  MoveC 4621 to (-315.82, 6.77, -76.56) mm, rotated rx -179.15 ry 0 rz -30.08 deg; joints [-3.162, -77.655, 137.613, -184.044, 59.828, 242.156] to (-316.49, 5.6, -77.12) mm, rotated rx -179.15 ry 0 rz -30.08 deg; joints [-3.197, -77.547, 137.594, -184.08, 59.918, 242.169]
  MoveL 4622 to (-316.49, 5.6, -77.12) mm, rotated rx -179.15 ry 0 rz -30.08 deg; joints [-3.197, -77.547, 137.594, -184.08, 59.918, 242.169]
  MoveC 4623 to (-316.55, 5.47, -77.12) mm, rotated rx -179.15 ry 0 rz -30.08 deg; joints [-3.2, -77.538, 137.596, -184.083, 59.93, 242.169] to (-316.58, 5.33, -77.12) mm, rotated rx -179.15 ry 0 rz -30.08 deg; joints [-3.201, -77.529, 137.599, -184.084, 59.942, 242.169]
  MoveL 4624 to (-316.58, 5.33, -77.12) mm, rotated rx -179.15 ry 0 rz -30.08 deg; joints [-3.201, -77.529, 137.599, -184.084, 59.942, 242.169]
  MoveC 4625 to (-316.6, 5.18, -77.12) mm, rotated rx -179.15 ry 0 rz -30.08 deg; joints [-3.203, -77.52, 137.602, -184.085, 59.954, 242.169] to (-316.66, 5.05, -77.12) mm, rotated rx -179.15 ry 0 rz -30.08 deg; joints [-3.206, -77.511, 137.604, -184.088, 59.965, 242.17]
  MoveL 4626 to (-316.66, 5.05, -77.12) mm, rotated rx -179.15 ry 0 rz -30.08 deg; joints [-3.206, -77.511, 137.604, -184.088, 59.965, 242.17]
  MoveL 4627 to (-327.16, -13.08, -77.12) mm, rotated rx -179.15 ry 0 rz -30.08 deg; joints [-3.765, -76.293, 137.92, -184.664, 61.515, 242.347]
  MoveC 4628 to (-327.25, -13.19, -77.12) mm, rotated rx -179.15 ry 0 rz -30.08 deg; joints [-3.77, -76.285, 137.921, -184.668, 61.524, 242.349] to (-327.36, -13.29, -77.12) mm, rotated rx -179.15 ry 0 rz -30.08 deg; joints [-3.776, -76.279, 137.923, -184.675, 61.532, 242.351]
  MoveL 4629 to (-327.36, -13.29, -77.12) mm, rotated rx -179.15 ry 0 rz -30.08 deg; joints [-3.776, -76.279, 137.923, -184.675, 61.532, 242.351]
  MoveC 4630 to (-327.47, -13.38, -77.12) mm, rotated rx -179.15 ry 0 rz -30.08 deg; joints [-3.781, -76.272, 137.924, -184.681, 61.54, 242.354] to (-327.55, -13.5, -77.12) mm, rotated rx -179.15 ry 0 rz -30.08 deg; joints [-3.786, -76.264, 137.926, -184.686, 61.55, 242.355]
  MoveL 4631 to (-327.55, -13.5, -77.12) mm, rotated rx -179.15 ry 0 rz -30.08 deg; joints [-3.786, -76.264, 137.926, -184.686, 61.55, 242.355]
  MoveC 4632 to (-328.23, -14.66, -77.67) mm, rotated rx -179.15 ry 0 rz -30.08 deg; joints [-3.82, -76.154, 137.904, -184.721, 61.639, 242.365] to (-328.51, -15.14, -79.02) mm, rotated rx -179.15 ry 0 rz -30.08 deg; joints [-3.83, -76.049, 137.812, -184.732, 61.654, 242.369]
  MoveL 4633 to (-328.51, -15.14, -79.02) mm, rotated rx -179.15 ry 0 rz -30.08 deg; joints [-3.83, -76.049, 137.812, -184.732, 61.654, 242.369]
  MoveL 4634 to (-328.51, -15.14, -81.56) mm, rotated rx -179.15 ry 0 rz -30.08 deg; joints [-3.821, -75.912, 137.626, -184.724, 61.604, 242.369]
  MoveC 4635 to (-328.23, -14.66, -82.91) mm, rotated rx -179.15 ry 0 rz -30.08 deg; joints [-3.802, -75.873, 137.52, -184.705, 61.536, 242.365] to (-327.55, -13.5, -83.46) mm, rotated rx -179.15 ry 0 rz -30.08 deg; joints [-3.764, -75.922, 137.46, -184.667, 61.426, 242.355]
  MoveL 4636 to (-327.55, -13.5, -83.46) mm, rotated rx -179.15 ry 0 rz -30.08 deg; joints [-3.764, -75.922, 137.46, -184.667, 61.426, 242.355]
  MoveC 4637 to (-327.47, -13.38, -83.46) mm, rotated rx -179.15 ry 0 rz -30.08 deg; joints [-3.76, -75.93, 137.458, -184.662, 61.417, 242.353] to (-327.36, -13.29, -83.46) mm, rotated rx -179.15 ry 0 rz -30.08 deg; joints [-3.754, -75.936, 137.457, -184.655, 61.409, 242.351]
  MoveL 4638 to (-327.36, -13.29, -83.46) mm, rotated rx -179.15 ry 0 rz -30.08 deg; joints [-3.754, -75.936, 137.457, -184.655, 61.409, 242.351]
  MoveC 4639 to (-327.25, -13.19, -83.46) mm, rotated rx -179.15 ry 0 rz -30.08 deg; joints [-3.748, -75.943, 137.456, -184.649, 61.401, 242.348] to (-327.16, -13.08, -83.46) mm, rotated rx -179.15 ry 0 rz -30.08 deg; joints [-3.743, -75.951, 137.454, -184.644, 61.391, 242.347]
  MoveL 4640 to (-327.16, -13.08, -83.46) mm, rotated rx -179.15 ry 0 rz -30.08 deg; joints [-3.743, -75.951, 137.454, -184.644, 61.391, 242.347]
  MoveL 4641 to (-316.66, 5.05, -83.46) mm, rotated rx -179.15 ry 0 rz -30.08 deg; joints [-3.187, -77.159, 137.141, -184.072, 59.853, 242.168]
  MoveC 4642 to (-316.6, 5.19, -83.46) mm, rotated rx -179.15 ry 0 rz -30.08 deg; joints [-3.184, -77.167, 137.138, -184.069, 59.842, 242.168] to (-316.58, 5.33, -83.46) mm, rotated rx -179.15 ry 0 rz -30.08 deg; joints [-3.183, -77.177, 137.135, -184.067, 59.83, 242.168]
  MoveL 4643 to (-316.58, 5.33, -83.46) mm, rotated rx -179.15 ry 0 rz -30.08 deg; joints [-3.183, -77.177, 137.135, -184.067, 59.83, 242.168]
  MoveC 4644 to (-316.55, 5.47, -83.46) mm, rotated rx -179.15 ry 0 rz -30.08 deg; joints [-3.181, -77.186, 137.132, -184.066, 59.818, 242.168] to (-316.49, 5.6, -83.46) mm, rotated rx -179.15 ry 0 rz -30.08 deg; joints [-3.178, -77.194, 137.13, -184.063, 59.807, 242.167]
  MoveL 4645 to (-316.49, 5.6, -83.46) mm, rotated rx -179.15 ry 0 rz -30.08 deg; joints [-3.178, -77.194, 137.13, -184.063, 59.807, 242.167]
  MoveC 4646 to (-315.82, 6.77, -84.02) mm, rotated rx -179.15 ry 0 rz -30.08 deg; joints [-3.141, -77.24, 137.068, -184.024, 59.698, 242.154] to (-315.54, 7.25, -85.37) mm, rotated rx -179.15 ry 0 rz -30.08 deg; joints [-3.122, -77.197, 136.96, -184.006, 59.633, 242.149]
  MoveL 4647 to (-315.54, 7.25, -85.37) mm, rotated rx -179.15 ry 0 rz -30.08 deg; joints [-3.122, -77.197, 136.96, -184.006, 59.633, 242.149]
  MoveL 4648 to (-315.54, 7.25, -87.91) mm, rotated rx -179.15 ry 0 rz -30.08 deg; joints [-3.115, -77.056, 136.774, -183.999, 59.588, 242.148]
  MoveC 4649 to (-315.82, 6.77, -89.26) mm, rotated rx -179.15 ry 0 rz -30.08 deg; joints [-3.126, -76.95, 136.685, -184.011, 59.605, 242.153] to (-316.49, 5.6, -89.81) mm, rotated rx -179.15 ry 0 rz -30.08 deg; joints [-3.16, -76.843, 136.665, -184.047, 59.693, 242.166]
  MoveL 4650 to (-316.49, 5.6, -89.81) mm, rotated rx -179.15 ry 0 rz -30.08 deg; joints [-3.16, -76.843, 136.665, -184.047, 59.693, 242.166]
  MoveC 4651 to (-316.55, 5.47, -89.81) mm, rotated rx -179.15 ry 0 rz -30.08 deg; joints [-3.163, -76.835, 136.668, -184.05, 59.704, 242.167] to (-316.58, 5.33, -89.81) mm, rotated rx -179.15 ry 0 rz -30.08 deg; joints [-3.165, -76.826, 136.67, -184.051, 59.716, 242.167]
  MoveL 4652 to (-316.58, 5.33, -89.81) mm, rotated rx -179.15 ry 0 rz -30.08 deg; joints [-3.165, -76.826, 136.67, -184.051, 59.716, 242.167]
  MoveC 4653 to (-316.6, 5.18, -89.81) mm, rotated rx -179.15 ry 0 rz -30.08 deg; joints [-3.166, -76.817, 136.673, -184.052, 59.728, 242.166] to (-316.66, 5.05, -89.81) mm, rotated rx -179.15 ry 0 rz -30.08 deg; joints [-3.169, -76.808, 136.676, -184.055, 59.739, 242.167]
  MoveL 4654 to (-316.66, 5.05, -89.81) mm, rotated rx -179.15 ry 0 rz -30.08 deg; joints [-3.169, -76.808, 136.676, -184.055, 59.739, 242.167]
  MoveL 4655 to (-327.16, -13.08, -89.81) mm, rotated rx -179.15 ry 0 rz -30.08 deg; joints [-3.722, -75.609, 136.987, -184.626, 61.265, 242.347]
  MoveC 4656 to (-327.25, -13.19, -89.81) mm, rotated rx -179.15 ry 0 rz -30.08 deg; joints [-3.727, -75.602, 136.989, -184.63, 61.274, 242.348] to (-327.36, -13.29, -89.81) mm, rotated rx -179.15 ry 0 rz -30.08 deg; joints [-3.732, -75.595, 136.99, -184.637, 61.282, 242.351]
  MoveL 4657 to (-327.36, -13.29, -89.81) mm, rotated rx -179.15 ry 0 rz -30.08 deg; joints [-3.732, -75.595, 136.99, -184.637, 61.282, 242.351]
  MoveC 4658 to (-327.47, -13.38, -89.81) mm, rotated rx -179.15 ry 0 rz -30.08 deg; joints [-3.738, -75.589, 136.991, -184.643, 61.29, 242.353] to (-327.55, -13.5, -89.81) mm, rotated rx -179.15 ry 0 rz -30.08 deg; joints [-3.743, -75.581, 136.993, -184.648, 61.3, 242.355]
  MoveL 4659 to (-327.55, -13.5, -89.81) mm, rotated rx -179.15 ry 0 rz -30.08 deg; joints [-3.743, -75.581, 136.993, -184.648, 61.3, 242.355]
  MoveC 4660 to (-328.23, -14.66, -90.37) mm, rotated rx -179.15 ry 0 rz -30.08 deg; joints [-3.776, -75.473, 136.97, -184.682, 61.387, 242.365] to (-328.51, -15.14, -91.72) mm, rotated rx -179.15 ry 0 rz -30.08 deg; joints [-3.786, -75.368, 136.879, -184.693, 61.4, 242.369]
  MoveL 4661 to (-328.51, -15.14, -91.72) mm, rotated rx -179.15 ry 0 rz -30.08 deg; joints [-3.786, -75.368, 136.879, -184.693, 61.4, 242.369]
  MoveL 4662 to (-328.51, -15.14, -94.26) mm, rotated rx -179.15 ry 0 rz -30.08 deg; joints [-3.778, -75.233, 136.691, -184.686, 61.348, 242.37]
  MoveC 4663 to (-328.23, -14.66, -95.6) mm, rotated rx -179.15 ry 0 rz -30.08 deg; joints [-3.759, -75.193, 136.584, -184.667, 61.28, 242.365] to (-327.55, -13.5, -96.16) mm, rotated rx -179.15 ry 0 rz -30.08 deg; joints [-3.721, -75.241, 136.525, -184.629, 61.171, 242.355]
  MoveL 4664 to (-327.55, -13.5, -96.16) mm, rotated rx -179.15 ry 0 rz -30.08 deg; joints [-3.721, -75.241, 136.525, -184.629, 61.171, 242.355]
  MoveC 4665 to (-327.47, -13.38, -96.16) mm, rotated rx -179.15 ry 0 rz -30.08 deg; joints [-3.717, -75.249, 136.523, -184.624, 61.161, 242.354] to (-327.36, -13.29, -96.16) mm, rotated rx -179.15 ry 0 rz -30.08 deg; joints [-3.711, -75.255, 136.522, -184.618, 61.154, 242.351]
  MoveL 4666 to (-327.36, -13.29, -96.16) mm, rotated rx -179.15 ry 0 rz -30.08 deg; joints [-3.711, -75.255, 136.522, -184.618, 61.154, 242.351]
  MoveC 4667 to (-327.25, -13.19, -96.16) mm, rotated rx -179.15 ry 0 rz -30.08 deg; joints [-3.705, -75.262, 136.52, -184.612, 61.146, 242.349] to (-327.16, -13.08, -96.16) mm, rotated rx -179.15 ry 0 rz -30.08 deg; joints [-3.701, -75.269, 136.519, -184.607, 61.136, 242.347]
  MoveL 4668 to (-327.16, -13.08, -96.16) mm, rotated rx -179.15 ry 0 rz -30.08 deg; joints [-3.701, -75.269, 136.519, -184.607, 61.136, 242.347]
  MoveL 4669 to (-316.66, 5.05, -96.16) mm, rotated rx -179.15 ry 0 rz -30.08 deg; joints [-3.151, -76.459, 136.21, -184.039, 59.622, 242.166]
  MoveC 4670 to (-316.6, 5.19, -96.16) mm, rotated rx -179.15 ry 0 rz -30.08 deg; joints [-3.148, -76.467, 136.207, -184.036, 59.611, 242.166] to (-316.58, 5.33, -96.16) mm, rotated rx -179.15 ry 0 rz -30.08 deg; joints [-3.147, -76.476, 136.204, -184.035, 59.599, 242.166]
  MoveL 4671 to (-316.58, 5.33, -96.16) mm, rotated rx -179.15 ry 0 rz -30.08 deg; joints [-3.147, -76.476, 136.204, -184.035, 59.599, 242.166]
  MoveC 4672 to (-316.55, 5.47, -96.16) mm, rotated rx -179.15 ry 0 rz -30.08 deg; joints [-3.145, -76.485, 136.202, -184.034, 59.587, 242.166] to (-316.49, 5.6, -96.16) mm, rotated rx -179.15 ry 0 rz -30.08 deg; joints [-3.142, -76.494, 136.199, -184.031, 59.576, 242.165]
  MoveL 4673 to (-316.49, 5.6, -96.16) mm, rotated rx -179.15 ry 0 rz -30.08 deg; joints [-3.142, -76.494, 136.199, -184.031, 59.576, 242.165]
  MoveC 4674 to (-315.82, 6.77, -96.72) mm, rotated rx -179.15 ry 0 rz -30.08 deg; joints [-3.105, -76.538, 136.137, -183.993, 59.468, 242.152] to (-315.54, 7.25, -98.07) mm, rotated rx -179.15 ry 0 rz -30.08 deg; joints [-3.087, -76.495, 136.029, -183.974, 59.403, 242.147]
  MoveL 4675 to (-315.54, 7.25, -98.07) mm, rotated rx -179.15 ry 0 rz -30.08 deg; joints [-3.087, -76.495, 136.029, -183.974, 59.403, 242.147]
  MoveL 4676 to (-315.54, 7.25, -100.61) mm, rotated rx -179.15 ry 0 rz -30.08 deg; joints [-3.08, -76.355, 135.842, -183.968, 59.356, 242.146]
  MoveC 4677 to (-315.82, 6.77, -101.95) mm, rotated rx -179.15 ry 0 rz -30.08 deg; joints [-3.091, -76.25, 135.752, -183.98, 59.37, 242.152] to (-316.49, 5.6, -102.51) mm, rotated rx -179.15 ry 0 rz -30.08 deg; joints [-3.125, -76.145, 135.732, -184.015, 59.457, 242.164]
  MoveL 4678 to (-316.49, 5.6, -102.51) mm, rotated rx -179.15 ry 0 rz -30.08 deg; joints [-3.125, -76.145, 135.732, -184.015, 59.457, 242.164]
  MoveC 4679 to (-316.55, 5.47, -102.51) mm, rotated rx -179.15 ry 0 rz -30.08 deg; joints [-3.128, -76.137, 135.734, -184.018, 59.468, 242.165] to (-316.58, 5.33, -102.51) mm, rotated rx -179.15 ry 0 rz -30.08 deg; joints [-3.129, -76.128, 135.737, -184.02, 59.479, 242.165]
  MoveL 4680 to (-316.58, 5.33, -102.51) mm, rotated rx -179.15 ry 0 rz -30.08 deg; joints [-3.129, -76.128, 135.737, -184.02, 59.479, 242.165]
  MoveC 4681 to (-316.6, 5.18, -102.51) mm, rotated rx -179.15 ry 0 rz -30.08 deg; joints [-3.13, -76.119, 135.74, -184.021, 59.491, 242.165] to (-316.66, 5.05, -102.51) mm, rotated rx -179.15 ry 0 rz -30.08 deg; joints [-3.133, -76.11, 135.742, -184.024, 59.502, 242.166]
  MoveL 4682 to (-316.66, 5.05, -102.51) mm, rotated rx -179.15 ry 0 rz -30.08 deg; joints [-3.133, -76.11, 135.742, -184.024, 59.502, 242.166]
  MoveL 4683 to (-327.16, -13.08, -102.51) mm, rotated rx -179.15 ry 0 rz -30.08 deg; joints [-3.68, -74.931, 136.049, -184.589, 61.005, 242.347]
  MoveC 4684 to (-327.25, -13.19, -102.51) mm, rotated rx -179.15 ry 0 rz -30.08 deg; joints [-3.684, -74.923, 136.051, -184.594, 61.015, 242.349] to (-327.36, -13.29, -102.51) mm, rotated rx -179.15 ry 0 rz -30.08 deg; joints [-3.69, -74.917, 136.052, -184.6, 61.023, 242.352]
  MoveL 4685 to (-327.36, -13.29, -102.51) mm, rotated rx -179.15 ry 0 rz -30.08 deg; joints [-3.69, -74.917, 136.052, -184.6, 61.023, 242.352]
  MoveC 4686 to (-327.47, -13.38, -102.51) mm, rotated rx -179.15 ry 0 rz -30.08 deg; joints [-3.696, -74.91, 136.053, -184.606, 61.03, 242.354] to (-327.55, -13.5, -102.51) mm, rotated rx -179.15 ry 0 rz -30.08 deg; joints [-3.7, -74.902, 136.055, -184.611, 61.04, 242.356]
  MoveL 4687 to (-327.55, -13.5, -102.51) mm, rotated rx -179.15 ry 0 rz -30.08 deg; joints [-3.7, -74.902, 136.055, -184.611, 61.04, 242.356]
  MoveC 4688 to (-328.23, -14.66, -103.07) mm, rotated rx -179.15 ry 0 rz -30.08 deg; joints [-3.734, -74.796, 136.032, -184.645, 61.125, 242.366] to (-328.51, -15.14, -104.42) mm, rotated rx -179.15 ry 0 rz -30.08 deg; joints [-3.744, -74.692, 135.94, -184.656, 61.136, 242.371]
  MoveL 4689 to (-328.51, -15.14, -104.42) mm, rotated rx -179.15 ry 0 rz -30.08 deg; joints [-3.744, -74.692, 135.94, -184.656, 61.136, 242.371]
  MoveL 4690 to (-328.51, -15.14, -106.95) mm, rotated rx -179.15 ry 0 rz -30.08 deg; joints [-3.735, -74.558, 135.752, -184.649, 61.082, 242.371]
  MoveC 4691 to (-328.23, -14.66, -108.3) mm, rotated rx -179.15 ry 0 rz -30.08 deg; joints [-3.716, -74.518, 135.644, -184.63, 61.014, 242.367] to (-327.55, -13.5, -108.86) mm, rotated rx -179.15 ry 0 rz -30.08 deg; joints [-3.68, -74.565, 135.585, -184.593, 60.906, 242.356]
  MoveL 4692 to (-327.55, -13.5, -108.86) mm, rotated rx -179.15 ry 0 rz -30.08 deg; joints [-3.68, -74.565, 135.585, -184.593, 60.906, 242.356]
  MoveC 4693 to (-327.47, -13.38, -108.86) mm, rotated rx -179.15 ry 0 rz -30.08 deg; joints [-3.675, -74.572, 135.583, -184.588, 60.897, 242.355] to (-327.36, -13.29, -108.86) mm, rotated rx -179.15 ry 0 rz -30.08 deg; joints [-3.669, -74.579, 135.582, -184.582, 60.889, 242.352]
  MoveL 4694 to (-327.36, -13.29, -108.86) mm, rotated rx -179.15 ry 0 rz -30.08 deg; joints [-3.669, -74.579, 135.582, -184.582, 60.889, 242.352]
  MoveC 4695 to (-327.25, -13.19, -108.86) mm, rotated rx -179.15 ry 0 rz -30.08 deg; joints [-3.664, -74.585, 135.58, -184.576, 60.881, 242.35] to (-327.16, -13.08, -108.86) mm, rotated rx -179.15 ry 0 rz -30.08 deg; joints [-3.659, -74.593, 135.579, -184.571, 60.872, 242.348]
  MoveL 4696 to (-327.16, -13.08, -108.86) mm, rotated rx -179.15 ry 0 rz -30.08 deg; joints [-3.659, -74.593, 135.579, -184.571, 60.872, 242.348]
  MoveL 4697 to (-316.66, 5.05, -108.86) mm, rotated rx -179.15 ry 0 rz -30.08 deg; joints [-3.116, -75.763, 135.273, -184.008, 59.38, 242.165]
  MoveC 4698 to (-316.6, 5.19, -108.86) mm, rotated rx -179.15 ry 0 rz -30.08 deg; joints [-3.113, -75.772, 135.271, -184.005, 59.369, 242.165] to (-316.58, 5.33, -108.86) mm, rotated rx -179.15 ry 0 rz -30.08 deg; joints [-3.112, -75.781, 135.268, -184.004, 59.358, 242.165]
  MoveL 4699 to (-316.58, 5.33, -108.86) mm, rotated rx -179.15 ry 0 rz -30.08 deg; joints [-3.112, -75.781, 135.268, -184.004, 59.358, 242.165]
  MoveC 4700 to (-316.55, 5.47, -108.86) mm, rotated rx -179.15 ry 0 rz -30.08 deg; joints [-3.11, -75.789, 135.266, -184.003, 59.346, 242.165] to (-316.49, 5.6, -108.86) mm, rotated rx -179.15 ry 0 rz -30.08 deg; joints [-3.107, -75.798, 135.263, -184, 59.335, 242.164]
  MoveL 4701 to (-316.49, 5.6, -108.86) mm, rotated rx -179.15 ry 0 rz -30.08 deg; joints [-3.107, -75.798, 135.263, -184, 59.335, 242.164]
  MoveC 4702 to (-315.82, 6.77, -109.42) mm, rotated rx -179.15 ry 0 rz -30.08 deg; joints [-3.071, -75.841, 135.201, -183.962, 59.228, 242.151] to (-315.54, 7.25, -110.76) mm, rotated rx -179.15 ry 0 rz -30.08 deg; joints [-3.053, -75.798, 135.092, -183.944, 59.163, 242.145]
  MoveL 4703 to (-315.54, 7.25, -110.76) mm, rotated rx -179.15 ry 0 rz -30.08 deg; joints [-3.053, -75.798, 135.092, -183.944, 59.163, 242.145]
  MoveL 4704 to (-315.54, 7.25, -113.3) mm, rotated rx -179.15 ry 0 rz -30.08 deg; joints [-3.046, -75.66, 134.905, -183.938, 59.113, 242.145]
  MoveC 4705 to (-315.82, 6.77, -114.65) mm, rotated rx -179.15 ry 0 rz -30.08 deg; joints [-3.057, -75.556, 134.814, -183.95, 59.127, 242.151] to (-316.49, 5.6, -115.21) mm, rotated rx -179.15 ry 0 rz -30.08 deg; joints [-3.09, -75.452, 134.793, -183.985, 59.211, 242.164]
  MoveL 4706 to (-316.49, 5.6, -115.21) mm, rotated rx -179.15 ry 0 rz -30.08 deg; joints [-3.09, -75.452, 134.793, -183.985, 59.211, 242.164]
  MoveC 4707 to (-316.55, 5.47, -115.21) mm, rotated rx -179.15 ry 0 rz -30.08 deg; joints [-3.093, -75.443, 134.796, -183.988, 59.222, 242.165] to (-316.58, 5.33, -115.21) mm, rotated rx -179.15 ry 0 rz -30.08 deg; joints [-3.094, -75.435, 134.798, -183.989, 59.233, 242.164]
  MoveL 4708 to (-316.58, 5.33, -115.21) mm, rotated rx -179.15 ry 0 rz -30.08 deg; joints [-3.094, -75.435, 134.798, -183.989, 59.233, 242.164]
  MoveC 4709 to (-316.6, 5.18, -115.21) mm, rotated rx -179.15 ry 0 rz -30.08 deg; joints [-3.096, -75.426, 134.801, -183.99, 59.245, 242.164] to (-316.66, 5.05, -115.21) mm, rotated rx -179.15 ry 0 rz -30.08 deg; joints [-3.098, -75.418, 134.804, -183.993, 59.256, 242.165]
  MoveL 4710 to (-316.66, 5.05, -115.21) mm, rotated rx -179.15 ry 0 rz -30.08 deg; joints [-3.098, -75.418, 134.804, -183.993, 59.256, 242.165]
  MoveL 4711 to (-327.16, -13.08, -115.21) mm, rotated rx -179.15 ry 0 rz -30.08 deg; joints [-3.639, -74.256, 135.107, -184.554, 60.737, 242.349]
  MoveC 4712 to (-327.25, -13.19, -115.21) mm, rotated rx -179.15 ry 0 rz -30.08 deg; joints [-3.643, -74.248, 135.109, -184.559, 60.746, 242.351] to (-327.36, -13.29, -115.21) mm, rotated rx -179.15 ry 0 rz -30.08 deg; joints [-3.649, -74.242, 135.11, -184.565, 60.754, 242.353]
  MoveL 4713 to (-327.36, -13.29, -115.21) mm, rotated rx -179.15 ry 0 rz -30.08 deg; joints [-3.649, -74.242, 135.11, -184.565, 60.754, 242.353]
  MoveC 4714 to (-327.47, -13.38, -115.21) mm, rotated rx -179.15 ry 0 rz -30.08 deg; joints [-3.655, -74.236, 135.111, -184.571, 60.761, 242.356] to (-327.55, -13.5, -115.21) mm, rotated rx -179.15 ry 0 rz -30.08 deg; joints [-3.659, -74.228, 135.113, -184.576, 60.771, 242.357]
  MoveL 4715 to (-327.55, -13.5, -115.21) mm, rotated rx -179.15 ry 0 rz -30.08 deg; joints [-3.659, -74.228, 135.113, -184.576, 60.771, 242.357]
  MoveC 4716 to (-328.23, -14.66, -115.77) mm, rotated rx -179.15 ry 0 rz -30.08 deg; joints [-3.692, -74.123, 135.089, -184.61, 60.854, 242.368] to (-328.51, -15.14, -117.11) mm, rotated rx -179.15 ry 0 rz -30.08 deg; joints [-3.702, -74.02, 134.996, -184.621, 60.864, 242.373]
  MoveL 4717 to (-328.51, -15.14, -117.11) mm, rotated rx -179.15 ry 0 rz -30.08 deg; joints [-3.702, -74.02, 134.996, -184.621, 60.864, 242.373]
  MoveL 4718 to (-328.51, -15.14, -119.65) mm, rotated rx -179.15 ry 0 rz -30.08 deg; joints [-3.694, -73.887, 134.807, -184.614, 60.808, 242.373]
  MoveC 4719 to (-328.23, -14.66, -121) mm, rotated rx -179.15 ry 0 rz -30.08 deg; joints [-3.675, -73.847, 134.699, -184.595, 60.739, 242.369] to (-327.55, -13.5, -121.56) mm, rotated rx -179.15 ry 0 rz -30.08 deg; joints [-3.639, -73.893, 134.64, -184.558, 60.633, 242.359]
  MoveL 4720 to (-327.55, -13.5, -121.56) mm, rotated rx -179.15 ry 0 rz -30.08 deg; joints [-3.639, -73.893, 134.64, -184.558, 60.633, 242.359]
  MoveC 4721 to (-327.47, -13.38, -121.56) mm, rotated rx -179.15 ry 0 rz -30.08 deg; joints [-3.634, -73.9, 134.638, -184.554, 60.624, 242.357] to (-327.36, -13.29, -121.56) mm, rotated rx -179.15 ry 0 rz -30.08 deg; joints [-3.629, -73.906, 134.637, -184.548, 60.616, 242.354]
  MoveL 4722 to (-327.36, -13.29, -121.56) mm, rotated rx -179.15 ry 0 rz -30.08 deg; joints [-3.629, -73.906, 134.637, -184.548, 60.616, 242.354]
  MoveC 4723 to (-327.25, -13.19, -121.56) mm, rotated rx -179.15 ry 0 rz -30.08 deg; joints [-3.623, -73.913, 134.636, -184.541, 60.608, 242.352] to (-327.16, -13.08, -121.56) mm, rotated rx -179.15 ry 0 rz -30.08 deg; joints [-3.619, -73.92, 134.634, -184.537, 60.599, 242.35]
  MoveL 4724 to (-327.16, -13.08, -121.56) mm, rotated rx -179.15 ry 0 rz -30.08 deg; joints [-3.619, -73.92, 134.634, -184.537, 60.599, 242.35]
  MoveL 4725 to (-316.66, 5.05, -121.56) mm, rotated rx -179.15 ry 0 rz -30.08 deg; joints [-3.081, -75.073, 134.332, -183.979, 59.129, 242.165]
  MoveC 4726 to (-316.6, 5.19, -121.56) mm, rotated rx -179.15 ry 0 rz -30.08 deg; joints [-3.078, -75.081, 134.33, -183.976, 59.118, 242.164] to (-316.58, 5.33, -121.56) mm, rotated rx -179.15 ry 0 rz -30.08 deg; joints [-3.077, -75.09, 134.327, -183.975, 59.107, 242.165]
  MoveL 4727 to (-316.58, 5.33, -121.56) mm, rotated rx -179.15 ry 0 rz -30.08 deg; joints [-3.077, -75.09, 134.327, -183.975, 59.107, 242.165]
  MoveC 4728 to (-316.55, 5.47, -121.56) mm, rotated rx -179.15 ry 0 rz -30.08 deg; joints [-3.076, -75.099, 134.324, -183.973, 59.095, 242.165] to (-316.49, 5.6, -121.56) mm, rotated rx -179.15 ry 0 rz -30.08 deg; joints [-3.073, -75.107, 134.322, -183.971, 59.084, 242.164]
  MoveL 4729 to (-316.49, 5.6, -121.56) mm, rotated rx -179.15 ry 0 rz -30.08 deg; joints [-3.073, -75.107, 134.322, -183.971, 59.084, 242.164]
  MoveC 4730 to (-315.82, 6.77, -122.11) mm, rotated rx -179.15 ry 0 rz -30.08 deg; joints [-3.037, -75.149, 134.26, -183.933, 58.979, 242.151] to (-315.54, 7.25, -123.46) mm, rotated rx -179.15 ry 0 rz -30.08 deg; joints [-3.019, -75.106, 134.151, -183.915, 58.912, 242.145]
  MoveL 4731 to (-315.54, 7.25, -123.46) mm, rotated rx -179.15 ry 0 rz -30.08 deg; joints [-3.019, -75.106, 134.151, -183.915, 58.912, 242.145]
  MoveL 4732 to (-315.54, 7.25, -126) mm, rotated rx -179.15 ry 0 rz -30.08 deg; joints [-3.012, -74.968, 133.962, -183.909, 58.861, 242.145]
  MoveC 4733 to (-315.82, 6.77, -127.35) mm, rotated rx -179.15 ry 0 rz -30.08 deg; joints [-3.023, -74.865, 133.87, -183.921, 58.873, 242.151] to (-316.49, 5.6, -127.91) mm, rotated rx -179.15 ry 0 rz -30.08 deg; joints [-3.056, -74.763, 133.85, -183.956, 58.956, 242.164]
  MoveL 4734 to (-316.49, 5.6, -127.91) mm, rotated rx -179.15 ry 0 rz -30.08 deg; joints [-3.056, -74.763, 133.85, -183.956, 58.956, 242.164]
  MoveC 4735 to (-316.55, 5.47, -127.91) mm, rotated rx -179.15 ry 0 rz -30.08 deg; joints [-3.059, -74.755, 133.852, -183.959, 58.966, 242.165] to (-316.58, 5.33, -127.91) mm, rotated rx -179.15 ry 0 rz -30.08 deg; joints [-3.06, -74.746, 133.855, -183.96, 58.978, 242.165]
  MoveL 4736 to (-316.58, 5.33, -127.91) mm, rotated rx -179.15 ry 0 rz -30.08 deg; joints [-3.06, -74.746, 133.855, -183.96, 58.978, 242.165]
  MoveC 4737 to (-316.6, 5.18, -127.91) mm, rotated rx -179.15 ry 0 rz -30.08 deg; joints [-3.061, -74.737, 133.857, -183.961, 58.989, 242.165] to (-316.66, 5.05, -127.91) mm, rotated rx -179.15 ry 0 rz -30.08 deg; joints [-3.064, -74.729, 133.86, -183.964, 59, 242.166]
  MoveL 4738 to (-316.66, 5.05, -127.91) mm, rotated rx -179.15 ry 0 rz -30.08 deg; joints [-3.064, -74.729, 133.86, -183.964, 59, 242.166]
  MoveL 4739 to (-327.16, -13.08, -127.91) mm, rotated rx -179.15 ry 0 rz -30.08 deg; joints [-3.599, -73.585, 134.159, -184.52, 60.459, 242.352]
  MoveC 4740 to (-327.25, -13.19, -127.91) mm, rotated rx -179.15 ry 0 rz -30.08 deg; joints [-3.603, -73.578, 134.161, -184.525, 60.468, 242.353] to (-327.36, -13.29, -127.91) mm, rotated rx -179.15 ry 0 rz -30.08 deg; joints [-3.609, -73.572, 134.162, -184.531, 60.476, 242.356]
  MoveL 4741 to (-327.36, -13.29, -127.91) mm, rotated rx -179.15 ry 0 rz -30.08 deg; joints [-3.609, -73.572, 134.162, -184.531, 60.476, 242.356]
  MoveC 4742 to (-327.47, -13.38, -127.91) mm, rotated rx -179.15 ry 0 rz -30.08 deg; joints [-3.614, -73.566, 134.164, -184.537, 60.483, 242.358] to (-327.55, -13.5, -127.91) mm, rotated rx -179.15 ry 0 rz -30.08 deg; joints [-3.619, -73.558, 134.165, -184.542, 60.493, 242.36]
  MoveL 4743 to (-327.55, -13.5, -127.91) mm, rotated rx -179.15 ry 0 rz -30.08 deg; joints [-3.619, -73.558, 134.165, -184.542, 60.493, 242.36]
  MoveC 4744 to (-328.23, -14.66, -128.46) mm, rotated rx -179.15 ry 0 rz -30.08 deg; joints [-3.651, -73.454, 134.141, -184.575, 60.574, 242.371] to (-328.51, -15.14, -129.81) mm, rotated rx -179.15 ry 0 rz -30.08 deg; joints [-3.661, -73.352, 134.048, -184.586, 60.582, 242.376]
  MoveL 4745 to (-328.51, -15.14, -129.81) mm, rotated rx -179.15 ry 0 rz -30.08 deg; joints [-3.661, -73.352, 134.048, -184.586, 60.582, 242.376]
  MoveL 4746 to (-328.51, -15.14, -132.35) mm, rotated rx -179.15 ry 0 rz -30.08 deg; joints [-3.653, -73.219, 133.858, -184.58, 60.525, 242.377]
  MoveC 4747 to (-328.23, -14.66, -133.7) mm, rotated rx -179.15 ry 0 rz -30.08 deg; joints [-3.635, -73.18, 133.749, -184.562, 60.456, 242.372] to (-327.55, -13.5, -134.25) mm, rotated rx -179.15 ry 0 rz -30.08 deg; joints [-3.599, -73.224, 133.69, -184.525, 60.351, 242.362]
  MoveL 4748 to (-327.55, -13.5, -134.25) mm, rotated rx -179.15 ry 0 rz -30.08 deg; joints [-3.599, -73.224, 133.69, -184.525, 60.351, 242.362]
  MoveC 4749 to (-327.47, -13.38, -134.25) mm, rotated rx -179.15 ry 0 rz -30.08 deg; joints [-3.594, -73.232, 133.688, -184.52, 60.341, 242.36] to (-327.36, -13.29, -134.25) mm, rotated rx -179.15 ry 0 rz -30.08 deg; joints [-3.589, -73.238, 133.687, -184.514, 60.334, 242.358]
  MoveL 4750 to (-327.36, -13.29, -134.25) mm, rotated rx -179.15 ry 0 rz -30.08 deg; joints [-3.589, -73.238, 133.687, -184.514, 60.334, 242.358]
  MoveC 4751 to (-327.25, -13.19, -134.25) mm, rotated rx -179.15 ry 0 rz -30.08 deg; joints [-3.583, -73.244, 133.686, -184.508, 60.326, 242.355] to (-327.16, -13.08, -134.25) mm, rotated rx -179.15 ry 0 rz -30.08 deg; joints [-3.579, -73.251, 133.684, -184.504, 60.317, 242.353]
  MoveL 4752 to (-327.16, -13.08, -134.25) mm, rotated rx -179.15 ry 0 rz -30.08 deg; joints [-3.579, -73.251, 133.684, -184.504, 60.317, 242.353]
  MoveL 4753 to (-316.66, 5.05, -134.25) mm, rotated rx -179.15 ry 0 rz -30.08 deg; joints [-3.048, -74.387, 133.386, -183.95, 58.868, 242.166]
  MoveC 4754 to (-316.6, 5.19, -134.25) mm, rotated rx -179.15 ry 0 rz -30.08 deg; joints [-3.045, -74.395, 133.384, -183.947, 58.858, 242.165] to (-316.58, 5.33, -134.25) mm, rotated rx -179.15 ry 0 rz -30.08 deg; joints [-3.043, -74.403, 133.381, -183.946, 58.846, 242.165]
  MoveL 4755 to (-316.58, 5.33, -134.25) mm, rotated rx -179.15 ry 0 rz -30.08 deg; joints [-3.043, -74.403, 133.381, -183.946, 58.846, 242.165]
  MoveC 4756 to (-316.55, 5.47, -134.25) mm, rotated rx -179.15 ry 0 rz -30.08 deg; joints [-3.042, -74.412, 133.378, -183.945, 58.835, 242.166] to (-316.49, 5.6, -134.25) mm, rotated rx -179.15 ry 0 rz -30.08 deg; joints [-3.039, -74.42, 133.376, -183.942, 58.824, 242.165]
  MoveL 4757 to (-316.49, 5.6, -134.25) mm, rotated rx -179.15 ry 0 rz -30.08 deg; joints [-3.039, -74.42, 133.376, -183.942, 58.824, 242.165]
  MoveC 4758 to (-315.82, 6.77, -134.81) mm, rotated rx -179.15 ry 0 rz -30.08 deg; joints [-3.004, -74.462, 133.314, -183.905, 58.72, 242.151] to (-315.54, 7.25, -136.16) mm, rotated rx -179.15 ry 0 rz -30.08 deg; joints [-2.986, -74.419, 133.204, -183.887, 58.653, 242.146]
  MoveL 4759 to (-315.54, 7.25, -136.16) mm, rotated rx -179.15 ry 0 rz -30.08 deg; joints [-2.986, -74.419, 133.204, -183.887, 58.653, 242.146]
  MoveL 4760 to (-315.54, 7.25, -138.7) mm, rotated rx -179.15 ry 0 rz -30.08 deg; joints [-2.979, -74.282, 133.014, -183.882, 58.6, 242.146]
  MoveC 4761 to (-315.82, 6.77, -140.05) mm, rotated rx -179.15 ry 0 rz -30.08 deg; joints [-2.99, -74.179, 132.922, -183.894, 58.61, 242.152] to (-316.49, 5.6, -140.6) mm, rotated rx -179.15 ry 0 rz -30.08 deg; joints [-3.023, -74.078, 132.901, -183.928, 58.691, 242.165]
  MoveL 4762 to (-316.49, 5.6, -140.6) mm, rotated rx -179.15 ry 0 rz -30.08 deg; joints [-3.023, -74.078, 132.901, -183.928, 58.691, 242.165]
  MoveC 4763 to (-316.55, 5.47, -140.6) mm, rotated rx -179.15 ry 0 rz -30.08 deg; joints [-3.026, -74.07, 132.903, -183.931, 58.701, 242.166] to (-316.58, 5.33, -140.6) mm, rotated rx -179.15 ry 0 rz -30.08 deg; joints [-3.027, -74.062, 132.906, -183.932, 58.713, 242.166]
  MoveL 4764 to (-316.58, 5.33, -140.6) mm, rotated rx -179.15 ry 0 rz -30.08 deg; joints [-3.027, -74.062, 132.906, -183.932, 58.713, 242.166]
  MoveC 4765 to (-316.6, 5.18, -140.6) mm, rotated rx -179.15 ry 0 rz -30.08 deg; joints [-3.028, -74.053, 132.908, -183.933, 58.724, 242.166] to (-316.66, 5.05, -140.6) mm, rotated rx -179.15 ry 0 rz -30.08 deg; joints [-3.031, -74.045, 132.911, -183.936, 58.734, 242.167]
  MoveL 4766 to (-316.66, 5.05, -140.6) mm, rotated rx -179.15 ry 0 rz -30.08 deg; joints [-3.031, -74.045, 132.911, -183.936, 58.734, 242.167]
  MoveL 4767 to (-327.16, -13.08, -140.6) mm, rotated rx -179.15 ry 0 rz -30.08 deg; joints [-3.559, -72.918, 133.207, -184.488, 60.173, 242.355]
  MoveC 4768 to (-327.25, -13.19, -140.6) mm, rotated rx -179.15 ry 0 rz -30.08 deg; joints [-3.564, -72.911, 133.209, -184.492, 60.182, 242.357] to (-327.36, -13.29, -140.6) mm, rotated rx -179.15 ry 0 rz -30.08 deg; joints [-3.569, -72.905, 133.21, -184.498, 60.19, 242.36]
  MoveL 4769 to (-327.36, -13.29, -140.6) mm, rotated rx -179.15 ry 0 rz -30.08 deg; joints [-3.569, -72.905, 133.21, -184.498, 60.19, 242.36]
  MoveC 4770 to (-327.47, -13.38, -140.6) mm, rotated rx -179.15 ry 0 rz -30.08 deg; joints [-3.575, -72.899, 133.211, -184.504, 60.197, 242.362] to (-327.55, -13.5, -140.6) mm, rotated rx -179.15 ry 0 rz -30.08 deg; joints [-3.579, -72.892, 133.213, -184.509, 60.206, 242.364]
  MoveL 4771 to (-327.55, -13.5, -140.6) mm, rotated rx -179.15 ry 0 rz -30.08 deg; joints [-3.579, -72.892, 133.213, -184.509, 60.206, 242.364]
  MoveC 4772 to (-328.23, -14.66, -141.16) mm, rotated rx -179.15 ry 0 rz -30.08 deg; joints [-3.611, -72.789, 133.188, -184.543, 60.286, 242.375] to (-328.51, -15.14, -142.51) mm, rotated rx -179.15 ry 0 rz -30.08 deg; joints [-3.621, -72.688, 133.094, -184.554, 60.293, 242.38]
  MoveL 4773 to (-328.51, -15.14, -142.51) mm, rotated rx -179.15 ry 0 rz -30.08 deg; joints [-3.621, -72.688, 133.094, -184.554, 60.293, 242.38]
  MoveL 4774 to (-328.51, -15.14, -145.05) mm, rotated rx -179.15 ry 0 rz -30.08 deg; joints [-3.613, -72.556, 132.903, -184.547, 60.234, 242.381]
  MoveC 4775 to (-328.23, -14.66, -146.39) mm, rotated rx -179.15 ry 0 rz -30.08 deg; joints [-3.595, -72.516, 132.794, -184.529, 60.164, 242.377] to (-327.55, -13.5, -146.95) mm, rotated rx -179.15 ry 0 rz -30.08 deg; joints [-3.56, -72.56, 132.735, -184.493, 60.06, 242.366]
  MoveL 4776 to (-327.55, -13.5, -146.95) mm, rotated rx -179.15 ry 0 rz -30.08 deg; joints [-3.56, -72.56, 132.735, -184.493, 60.06, 242.366]
  MoveC 4777 to (-327.47, -13.38, -146.95) mm, rotated rx -179.15 ry 0 rz -30.08 deg; joints [-3.555, -72.567, 132.733, -184.489, 60.051, 242.364] to (-327.36, -13.29, -146.95) mm, rotated rx -179.15 ry 0 rz -30.08 deg; joints [-3.55, -72.573, 132.732, -184.483, 60.043, 242.362]
  MoveL 4778 to (-327.36, -13.29, -146.95) mm, rotated rx -179.15 ry 0 rz -30.08 deg; joints [-3.55, -72.573, 132.732, -184.483, 60.043, 242.362]
  MoveC 4779 to (-327.25, -13.19, -146.95) mm, rotated rx -179.15 ry 0 rz -30.08 deg; joints [-3.544, -72.579, 132.731, -184.477, 60.036, 242.359] to (-327.16, -13.08, -146.95) mm, rotated rx -179.15 ry 0 rz -30.08 deg; joints [-3.54, -72.586, 132.729, -184.472, 60.027, 242.357]
  MoveL 4780 to (-327.16, -13.08, -146.95) mm, rotated rx -179.15 ry 0 rz -30.08 deg; joints [-3.54, -72.586, 132.729, -184.472, 60.027, 242.357]
  MoveL 4781 to (-316.66, 5.05, -146.95) mm, rotated rx -179.15 ry 0 rz -30.08 deg; joints [-3.015, -73.704, 132.434, -183.923, 58.598, 242.168]
  MoveC 4782 to (-316.6, 5.19, -146.95) mm, rotated rx -179.15 ry 0 rz -30.08 deg; joints [-3.012, -73.712, 132.432, -183.92, 58.588, 242.167] to (-316.58, 5.33, -146.95) mm, rotated rx -179.15 ry 0 rz -30.08 deg; joints [-3.011, -73.721, 132.429, -183.919, 58.577, 242.167]
  MoveL 4783 to (-316.58, 5.33, -146.95) mm, rotated rx -179.15 ry 0 rz -30.08 deg; joints [-3.011, -73.721, 132.429, -183.919, 58.577, 242.167]
  MoveC 4784 to (-316.55, 5.47, -146.95) mm, rotated rx -179.15 ry 0 rz -30.08 deg; joints [-3.009, -73.729, 132.427, -183.918, 58.566, 242.167] to (-316.49, 5.6, -146.95) mm, rotated rx -179.15 ry 0 rz -30.08 deg; joints [-3.006, -73.737, 132.424, -183.915, 58.555, 242.166]
  MoveL 4785 to (-316.49, 5.6, -146.95) mm, rotated rx -179.15 ry 0 rz -30.08 deg; joints [-3.006, -73.737, 132.424, -183.915, 58.555, 242.166]
  MoveC 4786 to (-315.82, 6.77, -147.51) mm, rotated rx -179.15 ry 0 rz -30.08 deg; joints [-2.971, -73.778, 132.362, -183.878, 58.451, 242.153] to (-315.54, 7.25, -148.86) mm, rotated rx -179.15 ry 0 rz -30.08 deg; joints [-2.954, -73.735, 132.252, -183.86, 58.384, 242.148]
  MoveL 4787 to (-315.54, 7.25, -148.86) mm, rotated rx -179.15 ry 0 rz -30.08 deg; joints [-2.954, -73.735, 132.252, -183.86, 58.384, 242.148]
  MoveL 4788 to (-315.54, 7.25, -151.4) mm, rotated rx -179.15 ry 0 rz -30.08 deg; joints [-2.947, -73.599, 132.061, -183.855, 58.329, 242.148]
  MoveC 4789 to (-315.82, 6.77, -152.74) mm, rotated rx -179.15 ry 0 rz -30.08 deg; joints [-2.958, -73.497, 131.968, -183.867, 58.338, 242.154] to (-316.49, 5.6, -153.3) mm, rotated rx -179.15 ry 0 rz -30.08 deg; joints [-2.99, -73.397, 131.947, -183.902, 58.417, 242.167]
  MoveL 4790 to (-316.49, 5.6, -153.3) mm, rotated rx -179.15 ry 0 rz -30.08 deg; joints [-2.99, -73.397, 131.947, -183.902, 58.417, 242.167]
  MoveC 4791 to (-316.55, 5.47, -153.3) mm, rotated rx -179.15 ry 0 rz -30.08 deg; joints [-2.993, -73.389, 131.949, -183.905, 58.428, 242.168] to (-316.58, 5.33, -153.3) mm, rotated rx -179.15 ry 0 rz -30.08 deg; joints [-2.994, -73.381, 131.952, -183.906, 58.439, 242.168]
  MoveL 4792 to (-316.58, 5.33, -153.3) mm, rotated rx -179.15 ry 0 rz -30.08 deg; joints [-2.994, -73.381, 131.952, -183.906, 58.439, 242.168]
  MoveC 4793 to (-316.6, 5.18, -153.3) mm, rotated rx -179.15 ry 0 rz -30.08 deg; joints [-2.996, -73.372, 131.954, -183.907, 58.45, 242.168] to (-316.66, 5.05, -153.3) mm, rotated rx -179.15 ry 0 rz -30.08 deg; joints [-2.998, -73.364, 131.957, -183.91, 58.46, 242.169]
  MoveL 4794 to (-316.66, 5.05, -153.3) mm, rotated rx -179.15 ry 0 rz -30.08 deg; joints [-2.998, -73.364, 131.957, -183.91, 58.46, 242.169]
  MoveL 4795 to (-327.16, -13.08, -153.3) mm, rotated rx -179.15 ry 0 rz -30.08 deg; joints [-3.521, -72.255, 132.249, -184.457, 59.878, 242.36]
  MoveC 4796 to (-327.25, -13.19, -153.3) mm, rotated rx -179.15 ry 0 rz -30.08 deg; joints [-3.525, -72.248, 132.251, -184.461, 59.887, 242.361] to (-327.36, -13.29, -153.3) mm, rotated rx -179.15 ry 0 rz -30.08 deg; joints [-3.531, -72.242, 132.252, -184.467, 59.895, 242.364]
  MoveL 4797 to (-327.36, -13.29, -153.3) mm, rotated rx -179.15 ry 0 rz -30.08 deg; joints [-3.531, -72.242, 132.252, -184.467, 59.895, 242.364]
  MoveC 4798 to (-327.47, -13.38, -153.3) mm, rotated rx -179.15 ry 0 rz -30.08 deg; joints [-3.536, -72.236, 132.253, -184.473, 59.902, 242.367] to (-327.55, -13.5, -153.3) mm, rotated rx -179.15 ry 0 rz -30.08 deg; joints [-3.54, -72.228, 132.255, -184.478, 59.911, 242.368]
  MoveL 4799 to (-327.55, -13.5, -153.3) mm, rotated rx -179.15 ry 0 rz -30.08 deg; joints [-3.54, -72.228, 132.255, -184.478, 59.911, 242.368]
  MoveC 4800 to (-328.23, -14.66, -153.86) mm, rotated rx -179.15 ry 0 rz -30.08 deg; joints [-3.572, -72.127, 132.23, -184.511, 59.989, 242.38] to (-328.51, -15.14, -155.21) mm, rotated rx -179.15 ry 0 rz -30.08 deg; joints [-3.582, -72.027, 132.135, -184.522, 59.994, 242.385]
  MoveL 4801 to (-328.51, -15.14, -155.21) mm, rotated rx -179.15 ry 0 rz -30.08 deg; joints [-3.582, -72.027, 132.135, -184.522, 59.994, 242.385]
  MoveL 4802 to (-328.51, -15.14, -157.74) mm, rotated rx -179.15 ry 0 rz -30.08 deg; joints [-3.574, -71.895, 131.943, -184.516, 59.934, 242.386]
  MoveC 4803 to (-328.23, -14.66, -159.09) mm, rotated rx -179.15 ry 0 rz -30.08 deg; joints [-3.557, -71.855, 131.834, -184.498, 59.864, 242.382] to (-327.55, -13.5, -159.65) mm, rotated rx -179.15 ry 0 rz -30.08 deg; joints [-3.521, -71.898, 131.774, -184.463, 59.76, 242.371]
  MoveL 4804 to (-327.55, -13.5, -159.65) mm, rotated rx -179.15 ry 0 rz -30.08 deg; joints [-3.521, -71.898, 131.774, -184.463, 59.76, 242.371]
  MoveC 4805 to (-327.47, -13.38, -159.65) mm, rotated rx -179.15 ry 0 rz -30.08 deg; joints [-3.517, -71.905, 131.773, -184.458, 59.752, 242.369] to (-327.36, -13.29, -159.65) mm, rotated rx -179.15 ry 0 rz -30.08 deg; joints [-3.512, -71.911, 131.771, -184.452, 59.744, 242.367]
  MoveL 4806 to (-327.36, -13.29, -159.65) mm, rotated rx -179.15 ry 0 rz -30.08 deg; joints [-3.512, -71.911, 131.771, -184.452, 59.744, 242.367]
  MoveC 4807 to (-327.25, -13.19, -159.65) mm, rotated rx -179.15 ry 0 rz -30.08 deg; joints [-3.506, -71.917, 131.77, -184.446, 59.737, 242.364] to (-327.16, -13.08, -159.65) mm, rotated rx -179.15 ry 0 rz -30.08 deg; joints [-3.502, -71.924, 131.769, -184.441, 59.728, 242.362]
  MoveL 4808 to (-327.16, -13.08, -159.65) mm, rotated rx -179.15 ry 0 rz -30.08 deg; joints [-3.502, -71.924, 131.769, -184.441, 59.728, 242.362]
  MoveL 4809 to (-316.66, 5.05, -159.65) mm, rotated rx -179.15 ry 0 rz -30.08 deg; joints [-2.982, -73.025, 131.477, -183.897, 58.32, 242.171]
  MoveC 4810 to (-316.6, 5.19, -159.65) mm, rotated rx -179.15 ry 0 rz -30.08 deg; joints [-2.98, -73.033, 131.475, -183.894, 58.309, 242.17] to (-316.58, 5.33, -159.65) mm, rotated rx -179.15 ry 0 rz -30.08 deg; joints [-2.978, -73.042, 131.472, -183.893, 58.298, 242.17]
  MoveL 4811 to (-316.58, 5.33, -159.65) mm, rotated rx -179.15 ry 0 rz -30.08 deg; joints [-2.978, -73.042, 131.472, -183.893, 58.298, 242.17]
  MoveC 4812 to (-316.55, 5.47, -159.65) mm, rotated rx -179.15 ry 0 rz -30.08 deg; joints [-2.977, -73.05, 131.47, -183.892, 58.287, 242.17] to (-316.49, 5.6, -159.65) mm, rotated rx -179.15 ry 0 rz -30.08 deg; joints [-2.974, -73.058, 131.467, -183.889, 58.277, 242.169]
  MoveL 4813 to (-316.49, 5.6, -159.65) mm, rotated rx -179.15 ry 0 rz -30.08 deg; joints [-2.974, -73.058, 131.467, -183.889, 58.277, 242.169]
  MoveC 4814 to (-315.82, 6.77, -160.21) mm, rotated rx -179.15 ry 0 rz -30.08 deg; joints [-2.939, -73.098, 131.405, -183.852, 58.174, 242.156] to (-315.54, 7.25, -161.55) mm, rotated rx -179.15 ry 0 rz -30.08 deg; joints [-2.922, -73.055, 131.295, -183.835, 58.107, 242.15]
  MoveL 4815 to (-315.54, 7.25, -161.55) mm, rotated rx -179.15 ry 0 rz -30.08 deg; joints [-2.922, -73.055, 131.295, -183.835, 58.107, 242.15]
  MoveL 4816 to (-315.54, 7.25, -164.09) mm, rotated rx -179.15 ry 0 rz -30.08 deg; joints [-2.916, -72.919, 131.103, -183.83, 58.05, 242.151]
  MoveC 4817 to (-315.82, 6.77, -165.44) mm, rotated rx -179.15 ry 0 rz -30.08 deg; joints [-2.927, -72.818, 131.009, -183.842, 58.057, 242.157] to (-316.49, 5.6, -166) mm, rotated rx -179.15 ry 0 rz -30.08 deg; joints [-2.958, -72.72, 130.987, -183.876, 58.135, 242.17]
  MoveL 4818 to (-316.49, 5.6, -166) mm, rotated rx -179.15 ry 0 rz -30.08 deg; joints [-2.958, -72.72, 130.987, -183.876, 58.135, 242.17]
  MoveC 4819 to (-316.55, 5.47, -166) mm, rotated rx -179.15 ry 0 rz -30.08 deg; joints [-2.961, -72.712, 130.989, -183.879, 58.145, 242.171] to (-316.58, 5.33, -166) mm, rotated rx -179.15 ry 0 rz -30.08 deg; joints [-2.963, -72.703, 130.992, -183.88, 58.156, 242.171]
  MoveL 4820 to (-316.58, 5.33, -166) mm, rotated rx -179.15 ry 0 rz -30.08 deg; joints [-2.963, -72.703, 130.992, -183.88, 58.156, 242.171]
  MoveC 4821 to (-316.6, 5.18, -166) mm, rotated rx -179.15 ry 0 rz -30.08 deg; joints [-2.964, -72.695, 130.995, -183.881, 58.167, 242.171] to (-316.66, 5.05, -166) mm, rotated rx -179.15 ry 0 rz -30.08 deg; joints [-2.967, -72.687, 130.997, -183.884, 58.177, 242.172]
  MoveL 4822 to (-316.66, 5.05, -166) mm, rotated rx -179.15 ry 0 rz -30.08 deg; joints [-2.967, -72.687, 130.997, -183.884, 58.177, 242.172]
  MoveL 4823 to (-327.16, -13.08, -166) mm, rotated rx -179.15 ry 0 rz -30.08 deg; joints [-3.483, -71.594, 131.286, -184.427, 59.576, 242.365]
  MoveC 4824 to (-327.25, -13.19, -166) mm, rotated rx -179.15 ry 0 rz -30.08 deg; joints [-3.488, -71.587, 131.288, -184.431, 59.584, 242.367] to (-327.36, -13.29, -166) mm, rotated rx -179.15 ry 0 rz -30.08 deg; joints [-3.493, -71.581, 131.289, -184.437, 59.592, 242.369]
  MoveL 4825 to (-327.36, -13.29, -166) mm, rotated rx -179.15 ry 0 rz -30.08 deg; joints [-3.493, -71.581, 131.289, -184.437, 59.592, 242.369]
  MoveC 4826 to (-327.47, -13.38, -166) mm, rotated rx -179.15 ry 0 rz -30.08 deg; joints [-3.498, -71.575, 131.29, -184.443, 59.599, 242.372] to (-327.55, -13.5, -166) mm, rotated rx -179.15 ry 0 rz -30.08 deg; joints [-3.503, -71.568, 131.292, -184.448, 59.608, 242.374]
  MoveL 4827 to (-327.55, -13.5, -166) mm, rotated rx -179.15 ry 0 rz -30.08 deg; joints [-3.503, -71.568, 131.292, -184.448, 59.608, 242.374]
  MoveC 4828 to (-328.23, -14.66, -166.56) mm, rotated rx -179.15 ry 0 rz -30.08 deg; joints [-3.534, -71.468, 131.267, -184.481, 59.684, 242.385] to (-328.51, -15.14, -167.9) mm, rotated rx -179.15 ry 0 rz -30.08 deg; joints [-3.544, -71.368, 131.171, -184.492, 59.688, 242.39]
  MoveL 4829 to (-328.51, -15.14, -167.9) mm, rotated rx -179.15 ry 0 rz -30.08 deg; joints [-3.544, -71.368, 131.171, -184.492, 59.688, 242.39]
  MoveL 4830 to (-328.51, -15.14, -170.44) mm, rotated rx -179.15 ry 0 rz -30.08 deg; joints [-3.536, -71.237, 130.978, -184.486, 59.626, 242.392]
  MoveC 4831 to (-328.23, -14.66, -171.79) mm, rotated rx -179.15 ry 0 rz -30.08 deg; joints [-3.519, -71.197, 130.868, -184.469, 59.556, 242.388] to (-327.55, -13.5, -172.35) mm, rotated rx -179.15 ry 0 rz -30.08 deg; joints [-3.484, -71.239, 130.809, -184.433, 59.453, 242.377]
  MoveL 4832 to (-327.55, -13.5, -172.35) mm, rotated rx -179.15 ry 0 rz -30.08 deg; joints [-3.484, -71.239, 130.809, -184.433, 59.453, 242.377]
  MoveC 4833 to (-327.47, -13.38, -172.35) mm, rotated rx -179.15 ry 0 rz -30.08 deg; joints [-3.48, -71.246, 130.807, -184.429, 59.444, 242.375] to (-327.36, -13.29, -172.35) mm, rotated rx -179.15 ry 0 rz -30.08 deg; joints [-3.474, -71.252, 130.806, -184.423, 59.437, 242.372]
  MoveL 4834 to (-327.36, -13.29, -172.35) mm, rotated rx -179.15 ry 0 rz -30.08 deg; joints [-3.474, -71.252, 130.806, -184.423, 59.437, 242.372]
  MoveC 4835 to (-327.25, -13.19, -172.35) mm, rotated rx -179.15 ry 0 rz -30.08 deg; joints [-3.469, -71.258, 130.805, -184.417, 59.43, 242.37] to (-327.16, -13.08, -172.35) mm, rotated rx -179.15 ry 0 rz -30.08 deg; joints [-3.465, -71.265, 130.803, -184.412, 59.421, 242.368]
  MoveL 4836 to (-327.16, -13.08, -172.35) mm, rotated rx -179.15 ry 0 rz -30.08 deg; joints [-3.465, -71.265, 130.803, -184.412, 59.421, 242.368]
  MoveL 4837 to (-316.66, 5.05, -172.35) mm, rotated rx -179.15 ry 0 rz -30.08 deg; joints [-2.951, -72.35, 130.515, -183.872, 58.032, 242.174]
  MoveC 4838 to (-316.6, 5.19, -172.35) mm, rotated rx -179.15 ry 0 rz -30.08 deg; joints [-2.948, -72.358, 130.513, -183.869, 58.022, 242.173] to (-316.58, 5.33, -172.35) mm, rotated rx -179.15 ry 0 rz -30.08 deg; joints [-2.947, -72.366, 130.51, -183.868, 58.011, 242.173]
  MoveL 4839 to (-316.58, 5.33, -172.35) mm, rotated rx -179.15 ry 0 rz -30.08 deg; joints [-2.947, -72.366, 130.51, -183.868, 58.011, 242.173]
  MoveC 4840 to (-316.55, 5.47, -172.35) mm, rotated rx -179.15 ry 0 rz -30.08 deg; joints [-2.946, -72.374, 130.507, -183.867, 58, 242.173] to (-316.49, 5.6, -172.35) mm, rotated rx -179.15 ry 0 rz -30.08 deg; joints [-2.943, -72.382, 130.505, -183.864, 57.99, 242.172]
  MoveL 4841 to (-316.49, 5.6, -172.35) mm, rotated rx -179.15 ry 0 rz -30.08 deg; joints [-2.943, -72.382, 130.505, -183.864, 57.99, 242.172]
  MoveC 4842 to (-315.82, 6.77, -172.9) mm, rotated rx -179.15 ry 0 rz -30.08 deg; joints [-2.908, -72.421, 130.443, -183.828, 57.888, 242.159] to (-315.54, 7.25, -174.25) mm, rotated rx -179.15 ry 0 rz -30.08 deg; joints [-2.891, -72.378, 130.332, -183.81, 57.82, 242.154]
  MoveL 4843 to (-315.54, 7.25, -174.25) mm, rotated rx -179.15 ry 0 rz -30.08 deg; joints [-2.891, -72.378, 130.332, -183.81, 57.82, 242.154]
  MoveL 4844 to (-315.54, 7.25, -176.79) mm, rotated rx -179.15 ry 0 rz -30.08 deg; joints [-2.885, -72.243, 130.139, -183.806, 57.762, 242.154]
  MoveC 4845 to (-315.82, 6.77, -178.14) mm, rotated rx -179.15 ry 0 rz -30.08 deg; joints [-2.896, -72.143, 130.045, -183.818, 57.768, 242.16] to (-316.49, 5.6, -178.7) mm, rotated rx -179.15 ry 0 rz -30.08 deg; joints [-2.927, -72.045, 130.022, -183.852, 57.844, 242.174]
  MoveL 4846 to (-316.49, 5.6, -178.7) mm, rotated rx -179.15 ry 0 rz -30.08 deg; joints [-2.927, -72.045, 130.022, -183.852, 57.844, 242.174]
  MoveC 4847 to (-316.55, 5.47, -178.7) mm, rotated rx -179.15 ry 0 rz -30.08 deg; joints [-2.93, -72.037, 130.024, -183.855, 57.854, 242.175] to (-316.58, 5.33, -178.7) mm, rotated rx -179.15 ry 0 rz -30.08 deg; joints [-2.931, -72.029, 130.027, -183.856, 57.864, 242.175]
  MoveL 4848 to (-316.58, 5.33, -178.7) mm, rotated rx -179.15 ry 0 rz -30.08 deg; joints [-2.931, -72.029, 130.027, -183.856, 57.864, 242.175]
  MoveC 4849 to (-316.6, 5.18, -178.7) mm, rotated rx -179.15 ry 0 rz -30.08 deg; joints [-2.933, -72.021, 130.029, -183.857, 57.875, 242.175] to (-316.66, 5.05, -178.7) mm, rotated rx -179.15 ry 0 rz -30.08 deg; joints [-2.935, -72.013, 130.032, -183.86, 57.885, 242.176]
  MoveL 4850 to (-316.66, 5.05, -178.7) mm, rotated rx -179.15 ry 0 rz -30.08 deg; joints [-2.935, -72.013, 130.032, -183.86, 57.885, 242.176]
  MoveL 4851 to (-327.16, -13.08, -178.7) mm, rotated rx -179.15 ry 0 rz -30.08 deg; joints [-3.447, -70.936, 130.318, -184.398, 59.265, 242.371]
  MoveC 4852 to (-327.25, -13.19, -178.7) mm, rotated rx -179.15 ry 0 rz -30.08 deg; joints [-3.451, -70.929, 130.32, -184.403, 59.273, 242.373] to (-327.36, -13.29, -178.7) mm, rotated rx -179.15 ry 0 rz -30.08 deg; joints [-3.456, -70.923, 130.321, -184.409, 59.281, 242.376]
  MoveL 4853 to (-327.36, -13.29, -178.7) mm, rotated rx -179.15 ry 0 rz -30.08 deg; joints [-3.456, -70.923, 130.321, -184.409, 59.281, 242.376]
  MoveC 4854 to (-327.47, -13.38, -178.7) mm, rotated rx -179.15 ry 0 rz -30.08 deg; joints [-3.461, -70.917, 130.322, -184.414, 59.288, 242.378] to (-327.55, -13.5, -178.7) mm, rotated rx -179.15 ry 0 rz -30.08 deg; joints [-3.466, -70.91, 130.324, -184.419, 59.297, 242.38]
  MoveL 4855 to (-327.55, -13.5, -178.7) mm, rotated rx -179.15 ry 0 rz -30.08 deg; joints [-3.466, -70.91, 130.324, -184.419, 59.297, 242.38]
  MoveC 4856 to (-328.23, -14.66, -179.25) mm, rotated rx -179.15 ry 0 rz -30.08 deg; joints [-3.497, -70.811, 130.298, -184.452, 59.371, 242.392] to (-328.51, -15.14, -180.6) mm, rotated rx -179.15 ry 0 rz -30.08 deg; joints [-3.507, -70.713, 130.202, -184.463, 59.374, 242.397]
  MoveL 4857 to (-328.51, -15.14, -180.6) mm, rotated rx -179.15 ry 0 rz -30.08 deg; joints [-3.507, -70.713, 130.202, -184.463, 59.374, 242.397]
  MoveL 4858 to (-328.51, -15.14, -183.14) mm, rotated rx -179.15 ry 0 rz -30.08 deg; joints [-3.499, -70.582, 130.008, -184.457, 59.31, 242.398]
  MoveC 4859 to (-328.23, -14.66, -184.49) mm, rotated rx -179.15 ry 0 rz -30.08 deg; joints [-3.482, -70.542, 129.897, -184.44, 59.24, 242.394] to (-327.55, -13.5, -185.04) mm, rotated rx -179.15 ry 0 rz -30.08 deg; joints [-3.447, -70.583, 129.837, -184.405, 59.138, 242.383]
  MoveL 4860 to (-327.55, -13.5, -185.04) mm, rotated rx -179.15 ry 0 rz -30.08 deg; joints [-3.447, -70.583, 129.837, -184.405, 59.138, 242.383]
  MoveC 4861 to (-327.47, -13.38, -185.04) mm, rotated rx -179.15 ry 0 rz -30.08 deg; joints [-3.443, -70.59, 129.836, -184.401, 59.129, 242.381] to (-327.36, -13.29, -185.04) mm, rotated rx -179.15 ry 0 rz -30.08 deg; joints [-3.438, -70.595, 129.835, -184.395, 59.122, 242.379]
  MoveL 4862 to (-327.36, -13.29, -185.04) mm, rotated rx -179.15 ry 0 rz -30.08 deg; joints [-3.438, -70.595, 129.835, -184.395, 59.122, 242.379]
  MoveC 4863 to (-327.25, -13.19, -185.04) mm, rotated rx -179.15 ry 0 rz -30.08 deg; joints [-3.433, -70.601, 129.834, -184.389, 59.115, 242.376] to (-327.16, -13.08, -185.04) mm, rotated rx -179.15 ry 0 rz -30.08 deg; joints [-3.428, -70.608, 129.832, -184.384, 59.106, 242.375]
  MoveL 4864 to (-327.16, -13.08, -185.04) mm, rotated rx -179.15 ry 0 rz -30.08 deg; joints [-3.428, -70.608, 129.832, -184.384, 59.106, 242.375]
  MoveL 4865 to (-316.66, 5.05, -185.04) mm, rotated rx -179.15 ry 0 rz -30.08 deg; joints [-2.92, -71.678, 129.547, -183.848, 57.736, 242.178]
  MoveC 4866 to (-316.6, 5.19, -185.04) mm, rotated rx -179.15 ry 0 rz -30.08 deg; joints [-2.917, -71.685, 129.545, -183.845, 57.726, 242.177] to (-316.58, 5.33, -185.04) mm, rotated rx -179.15 ry 0 rz -30.08 deg; joints [-2.916, -71.693, 129.542, -183.844, 57.716, 242.177]
  MoveL 4867 to (-316.58, 5.33, -185.04) mm, rotated rx -179.15 ry 0 rz -30.08 deg; joints [-2.916, -71.693, 129.542, -183.844, 57.716, 242.177]
  MoveC 4868 to (-316.55, 5.47, -185.04) mm, rotated rx -179.15 ry 0 rz -30.08 deg; joints [-2.915, -71.701, 129.539, -183.843, 57.705, 242.177] to (-316.49, 5.6, -185.04) mm, rotated rx -179.15 ry 0 rz -30.08 deg; joints [-2.912, -71.709, 129.537, -183.84, 57.695, 242.176]
  MoveL 4869 to (-316.49, 5.6, -185.04) mm, rotated rx -179.15 ry 0 rz -30.08 deg; joints [-2.912, -71.709, 129.537, -183.84, 57.695, 242.176]
  MoveC 4870 to (-315.82, 6.77, -185.6) mm, rotated rx -179.15 ry 0 rz -30.08 deg; joints [-2.878, -71.747, 129.475, -183.804, 57.593, 242.163] to (-315.54, 7.25, -186.95) mm, rotated rx -179.15 ry 0 rz -30.08 deg; joints [-2.861, -71.704, 129.364, -183.787, 57.525, 242.158]
  MoveL 4871 to (-315.54, 7.25, -186.95) mm, rotated rx -179.15 ry 0 rz -30.08 deg; joints [-2.861, -71.704, 129.364, -183.787, 57.525, 242.158]
  MoveL 4872 to (-315.54, 7.25, -189.49) mm, rotated rx -179.15 ry 0 rz -30.08 deg; joints [-2.855, -71.569, 129.169, -183.783, 57.465, 242.159]
  MoveC 4873 to (-315.82, 6.77, -190.84) mm, rotated rx -179.15 ry 0 rz -30.08 deg; joints [-2.866, -71.47, 129.074, -183.795, 57.47, 242.165] to (-316.49, 5.6, -191.39) mm, rotated rx -179.15 ry 0 rz -30.08 deg; joints [-2.897, -71.374, 129.051, -183.828, 57.544, 242.179]
  MoveL 4874 to (-316.49, 5.6, -191.39) mm, rotated rx -179.15 ry 0 rz -30.08 deg; joints [-2.897, -71.374, 129.051, -183.828, 57.544, 242.179]
  MoveC 4875 to (-316.55, 5.47, -191.39) mm, rotated rx -179.15 ry 0 rz -30.08 deg; joints [-2.9, -71.366, 129.053, -183.831, 57.554, 242.18] to (-316.58, 5.33, -191.39) mm, rotated rx -179.15 ry 0 rz -30.08 deg; joints [-2.901, -71.358, 129.056, -183.832, 57.565, 242.18]
  MoveL 4876 to (-316.58, 5.33, -191.39) mm, rotated rx -179.15 ry 0 rz -30.08 deg; joints [-2.901, -71.358, 129.056, -183.832, 57.565, 242.18]
  MoveC 4877 to (-316.6, 5.18, -191.39) mm, rotated rx -179.15 ry 0 rz -30.08 deg; joints [-2.902, -71.35, 129.059, -183.833, 57.575, 242.18] to (-316.66, 5.05, -191.39) mm, rotated rx -179.15 ry 0 rz -30.08 deg; joints [-2.905, -71.342, 129.061, -183.836, 57.585, 242.181]
  MoveL 4878 to (-316.66, 5.05, -191.39) mm, rotated rx -179.15 ry 0 rz -30.08 deg; joints [-2.905, -71.342, 129.061, -183.836, 57.585, 242.181]
  MoveL 4879 to (-327.16, -13.08, -191.39) mm, rotated rx -179.15 ry 0 rz -30.08 deg; joints [-3.411, -70.281, 129.344, -184.371, 58.946, 242.378]
  MoveC 4880 to (-327.25, -13.19, -191.39) mm, rotated rx -179.15 ry 0 rz -30.08 deg; joints [-3.415, -70.274, 129.346, -184.375, 58.955, 242.38] to (-327.36, -13.29, -191.39) mm, rotated rx -179.15 ry 0 rz -30.08 deg; joints [-3.42, -70.268, 129.347, -184.381, 58.962, 242.382]
  MoveL 4881 to (-327.36, -13.29, -191.39) mm, rotated rx -179.15 ry 0 rz -30.08 deg; joints [-3.42, -70.268, 129.347, -184.381, 58.962, 242.382]
  MoveC 4882 to (-327.47, -13.38, -191.39) mm, rotated rx -179.15 ry 0 rz -30.08 deg; joints [-3.425, -70.262, 129.348, -184.387, 58.969, 242.385] to (-327.55, -13.5, -191.39) mm, rotated rx -179.15 ry 0 rz -30.08 deg; joints [-3.429, -70.255, 129.35, -184.391, 58.977, 242.387]
  MoveL 4883 to (-327.55, -13.5, -191.39) mm, rotated rx -179.15 ry 0 rz -30.08 deg; joints [-3.429, -70.255, 129.35, -184.391, 58.977, 242.387]
  MoveC 4884 to (-328.23, -14.66, -191.95) mm, rotated rx -179.15 ry 0 rz -30.08 deg; joints [-3.46, -70.157, 129.324, -184.424, 59.05, 242.399] to (-328.51, -15.14, -193.3) mm, rotated rx -179.15 ry 0 rz -30.08 deg; joints [-3.47, -70.059, 129.227, -184.435, 59.052, 242.404]
  MoveL 4885 to (-328.51, -15.14, -193.3) mm, rotated rx -179.15 ry 0 rz -30.08 deg; joints [-3.47, -70.059, 129.227, -184.435, 59.052, 242.404]
  MoveL 4886 to (-328.51, -15.14, -195.84) mm, rotated rx -179.15 ry 0 rz -30.08 deg; joints [-3.463, -69.929, 129.031, -184.43, 58.987, 242.406]
  MoveC 4887 to (-328.23, -14.66, -197.18) mm, rotated rx -179.15 ry 0 rz -30.08 deg; joints [-3.446, -69.888, 128.921, -184.413, 58.916, 242.402] to (-327.55, -13.5, -197.74) mm, rotated rx -179.15 ry 0 rz -30.08 deg; joints [-3.412, -69.929, 128.861, -184.378, 58.815, 242.391]
  MoveL 4888 to (-327.55, -13.5, -197.74) mm, rotated rx -179.15 ry 0 rz -30.08 deg; joints [-3.412, -69.929, 128.861, -184.378, 58.815, 242.391]
  MoveC 4889 to (-327.47, -13.38, -197.74) mm, rotated rx -179.15 ry 0 rz -30.08 deg; joints [-3.408, -69.935, 128.859, -184.374, 58.806, 242.389] to (-327.36, -13.29, -197.74) mm, rotated rx -179.15 ry 0 rz -30.08 deg; joints [-3.402, -69.941, 128.858, -184.368, 58.799, 242.386]
  MoveL 4890 to (-327.36, -13.29, -197.74) mm, rotated rx -179.15 ry 0 rz -30.08 deg; joints [-3.402, -69.941, 128.858, -184.368, 58.799, 242.386]
  MoveC 4891 to (-327.25, -13.19, -197.74) mm, rotated rx -179.15 ry 0 rz -30.08 deg; joints [-3.397, -69.947, 128.857, -184.362, 58.792, 242.384] to (-327.16, -13.08, -197.74) mm, rotated rx -179.15 ry 0 rz -30.08 deg; joints [-3.393, -69.954, 128.855, -184.358, 58.784, 242.382]
  MoveL 4892 to (-327.16, -13.08, -197.74) mm, rotated rx -179.15 ry 0 rz -30.08 deg; joints [-3.393, -69.954, 128.855, -184.358, 58.784, 242.382]
  MoveL 4893 to (-316.66, 5.05, -197.74) mm, rotated rx -179.15 ry 0 rz -30.08 deg; joints [-2.89, -71.008, 128.573, -183.825, 57.432, 242.183]
  MoveC 4894 to (-316.6, 5.19, -197.74) mm, rotated rx -179.15 ry 0 rz -30.08 deg; joints [-2.887, -71.015, 128.571, -183.822, 57.422, 242.182] to (-316.58, 5.33, -197.74) mm, rotated rx -179.15 ry 0 rz -30.08 deg; joints [-2.886, -71.023, 128.568, -183.821, 57.412, 242.182]
  MoveL 4895 to (-316.58, 5.33, -197.74) mm, rotated rx -179.15 ry 0 rz -30.08 deg; joints [-2.886, -71.023, 128.568, -183.821, 57.412, 242.182]
  MoveC 4896 to (-316.55, 5.47, -197.74) mm, rotated rx -179.15 ry 0 rz -30.08 deg; joints [-2.885, -71.031, 128.566, -183.82, 57.401, 242.182] to (-316.49, 5.6, -197.74) mm, rotated rx -179.15 ry 0 rz -30.08 deg; joints [-2.882, -71.039, 128.564, -183.817, 57.391, 242.181]
  MoveL 4897 to (-316.49, 5.6, -197.74) mm, rotated rx -179.15 ry 0 rz -30.08 deg; joints [-2.882, -71.039, 128.564, -183.817, 57.391, 242.181]
  MoveC 4898 to (-315.82, 6.77, -198.3) mm, rotated rx -179.15 ry 0 rz -30.08 deg; joints [-2.848, -71.076, 128.501, -183.782, 57.291, 242.168] to (-315.54, 7.25, -199.65) mm, rotated rx -179.15 ry 0 rz -30.08 deg; joints [-2.832, -71.032, 128.389, -183.765, 57.222, 242.163]
  MoveL 4899 to (-315.54, 7.25, -199.65) mm, rotated rx -179.15 ry 0 rz -30.08 deg; joints [-2.832, -71.032, 128.389, -183.765, 57.222, 242.163]
  MoveL 4900 to (-315.54, 7.25, -202.19) mm, rotated rx -179.15 ry 0 rz -30.08 deg; joints [-2.826, -70.899, 128.194, -183.76, 57.16, 242.164]
  MoveC 4901 to (-315.82, 6.77, -203.53) mm, rotated rx -179.15 ry 0 rz -30.08 deg; joints [-2.836, -70.8, 128.098, -183.773, 57.163, 242.17] to (-316.49, 5.6, -204.09) mm, rotated rx -179.15 ry 0 rz -30.08 deg; joints [-2.867, -70.704, 128.075, -183.806, 57.236, 242.184]
  MoveL 4902 to (-316.49, 5.6, -204.09) mm, rotated rx -179.15 ry 0 rz -30.08 deg; joints [-2.867, -70.704, 128.075, -183.806, 57.236, 242.184]
  MoveC 4903 to (-316.55, 5.47, -204.09) mm, rotated rx -179.15 ry 0 rz -30.08 deg; joints [-2.87, -70.697, 128.077, -183.809, 57.246, 242.185] to (-316.58, 5.33, -204.09) mm, rotated rx -179.15 ry 0 rz -30.08 deg; joints [-2.871, -70.689, 128.079, -183.81, 57.257, 242.185]
  MoveL 4904 to (-316.58, 5.33, -204.09) mm, rotated rx -179.15 ry 0 rz -30.08 deg; joints [-2.871, -70.689, 128.079, -183.81, 57.257, 242.185]
  MoveC 4905 to (-316.6, 5.18, -204.09) mm, rotated rx -179.15 ry 0 rz -30.08 deg; joints [-2.872, -70.681, 128.082, -183.811, 57.267, 242.185] to (-316.66, 5.05, -204.09) mm, rotated rx -179.15 ry 0 rz -30.08 deg; joints [-2.875, -70.674, 128.084, -183.814, 57.277, 242.186]
  MoveL 4906 to (-316.66, 5.05, -204.09) mm, rotated rx -179.15 ry 0 rz -30.08 deg; joints [-2.875, -70.674, 128.084, -183.814, 57.277, 242.186]
  MoveL 4907 to (-327.16, -13.08, -204.09) mm, rotated rx -179.15 ry 0 rz -30.08 deg; joints [-3.375, -69.627, 128.365, -184.345, 58.62, 242.386]
  MoveC 4908 to (-327.25, -13.19, -204.09) mm, rotated rx -179.15 ry 0 rz -30.08 deg; joints [-3.379, -69.62, 128.367, -184.349, 58.628, 242.388] to (-327.36, -13.29, -204.09) mm, rotated rx -179.15 ry 0 rz -30.08 deg; joints [-3.385, -69.615, 128.368, -184.355, 58.635, 242.39]
  MoveL 4909 to (-327.36, -13.29, -204.09) mm, rotated rx -179.15 ry 0 rz -30.08 deg; joints [-3.385, -69.615, 128.368, -184.355, 58.635, 242.39]
  MoveC 4910 to (-327.47, -13.38, -204.09) mm, rotated rx -179.15 ry 0 rz -30.08 deg; joints [-3.39, -69.609, 128.369, -184.361, 58.642, 242.393] to (-327.55, -13.5, -204.09) mm, rotated rx -179.15 ry 0 rz -30.08 deg; joints [-3.394, -69.602, 128.37, -184.365, 58.651, 242.395]
  MoveL 4911 to (-327.55, -13.5, -204.09) mm, rotated rx -179.15 ry 0 rz -30.08 deg; joints [-3.394, -69.602, 128.37, -184.365, 58.651, 242.395]
  MoveC 4912 to (-328.23, -14.66, -204.65) mm, rotated rx -179.15 ry 0 rz -30.08 deg; joints [-3.425, -69.505, 128.344, -184.398, 58.722, 242.407] to (-328.51, -15.14, -206) mm, rotated rx -179.15 ry 0 rz -30.08 deg; joints [-3.434, -69.408, 128.247, -184.409, 58.722, 242.413]
  MoveL 4913 to (-328.51, -15.14, -206) mm, rotated rx -179.15 ry 0 rz -30.08 deg; joints [-3.434, -69.408, 128.247, -184.409, 58.722, 242.413]
  MoveL 4914 to (-328.51, -15.14, -208.53) mm, rotated rx -179.15 ry 0 rz -30.08 deg; joints [-3.427, -69.278, 128.05, -184.404, 58.655, 242.414]
  MoveC 4915 to (-328.23, -14.66, -209.88) mm, rotated rx -179.15 ry 0 rz -30.08 deg; joints [-3.41, -69.237, 127.938, -184.387, 58.585, 242.41] to (-327.55, -13.5, -210.44) mm, rotated rx -179.15 ry 0 rz -30.08 deg; joints [-3.377, -69.276, 127.879, -184.352, 58.484, 242.399]
  MoveL 4916 to (-327.55, -13.5, -210.44) mm, rotated rx -179.15 ry 0 rz -30.08 deg; joints [-3.377, -69.276, 127.879, -184.352, 58.484, 242.399]
  MoveC 4917 to (-327.47, -13.38, -210.44) mm, rotated rx -179.15 ry 0 rz -30.08 deg; joints [-3.373, -69.283, 127.877, -184.348, 58.476, 242.397] to (-327.36, -13.29, -210.44) mm, rotated rx -179.15 ry 0 rz -30.08 deg; joints [-3.367, -69.289, 127.876, -184.342, 58.469, 242.394]
  MoveL 4918 to (-327.36, -13.29, -210.44) mm, rotated rx -179.15 ry 0 rz -30.08 deg; joints [-3.367, -69.289, 127.876, -184.342, 58.469, 242.394]
  MoveC 4919 to (-327.25, -13.19, -210.44) mm, rotated rx -179.15 ry 0 rz -30.08 deg; joints [-3.362, -69.294, 127.875, -184.336, 58.462, 242.392] to (-327.16, -13.08, -210.44) mm, rotated rx -179.15 ry 0 rz -30.08 deg; joints [-3.358, -69.301, 127.873, -184.332, 58.454, 242.39]
  MoveL 4920 to (-327.16, -13.08, -210.44) mm, rotated rx -179.15 ry 0 rz -30.08 deg; joints [-3.358, -69.301, 127.873, -184.332, 58.454, 242.39]
  MoveL 4921 to (-316.66, 5.05, -210.44) mm, rotated rx -179.15 ry 0 rz -30.08 deg; joints [-2.86, -70.34, 127.594, -183.803, 57.12, 242.189]
  MoveC 4922 to (-316.6, 5.19, -210.44) mm, rotated rx -179.15 ry 0 rz -30.08 deg; joints [-2.858, -70.348, 127.592, -183.8, 57.11, 242.188] to (-316.58, 5.33, -210.44) mm, rotated rx -179.15 ry 0 rz -30.08 deg; joints [-2.856, -70.356, 127.589, -183.799, 57.1, 242.188]
  MoveL 4923 to (-316.58, 5.33, -210.44) mm, rotated rx -179.15 ry 0 rz -30.08 deg; joints [-2.856, -70.355, 127.589, -183.799, 57.1, 242.188]
  MoveC 4924 to (-316.55, 5.47, -210.44) mm, rotated rx -179.15 ry 0 rz -30.08 deg; joints [-2.855, -70.363, 127.586, -183.798, 57.089, 242.188] to (-316.49, 5.6, -210.44) mm, rotated rx -179.15 ry 0 rz -30.08 deg; joints [-2.852, -70.371, 127.584, -183.795, 57.079, 242.187]
  MoveL 4925 to (-316.49, 5.6, -210.44) mm, rotated rx -179.15 ry 0 rz -30.08 deg; joints [-2.852, -70.371, 127.584, -183.795, 57.079, 242.187]
  MoveC 4926 to (-315.82, 6.77, -211) mm, rotated rx -179.15 ry 0 rz -30.08 deg; joints [-2.819, -70.407, 127.522, -183.76, 56.98, 242.173] to (-315.54, 7.25, -212.34) mm, rotated rx -179.15 ry 0 rz -30.08 deg; joints [-2.803, -70.364, 127.41, -183.744, 56.91, 242.168]
  MoveL 4927 to (-315.54, 7.25, -212.34) mm, rotated rx -179.15 ry 0 rz -30.08 deg; joints [-2.803, -70.364, 127.41, -183.744, 56.91, 242.168]
  MoveL 4928 to (-315.54, 7.25, -214.88) mm, rotated rx -179.15 ry 0 rz -30.08 deg; joints [-2.797, -70.23, 127.213, -183.739, 56.847, 242.169]
  MoveC 4929 to (-315.82, 6.77, -216.23) mm, rotated rx -179.15 ry 0 rz -30.08 deg; joints [-2.807, -70.132, 127.116, -183.752, 56.849, 242.176] to (-316.49, 5.6, -216.79) mm, rotated rx -179.15 ry 0 rz -30.08 deg; joints [-2.838, -70.038, 127.092, -183.785, 56.92, 242.19]
  MoveL 4930 to (-316.49, 5.6, -216.79) mm, rotated rx -179.15 ry 0 rz -30.08 deg; joints [-2.838, -70.038, 127.092, -183.785, 56.92, 242.19]
  MoveC 4931 to (-316.55, 5.47, -216.79) mm, rotated rx -179.15 ry 0 rz -30.08 deg; joints [-2.841, -70.03, 127.095, -183.788, 56.93, 242.191] to (-316.58, 5.33, -216.79) mm, rotated rx -179.15 ry 0 rz -30.08 deg; joints [-2.842, -70.022, 127.097, -183.789, 56.94, 242.191]
  MoveL 4932 to (-316.58, 5.33, -216.79) mm, rotated rx -179.15 ry 0 rz -30.08 deg; joints [-2.842, -70.022, 127.097, -183.789, 56.94, 242.191]
  MoveC 4933 to (-316.6, 5.18, -216.79) mm, rotated rx -179.15 ry 0 rz -30.08 deg; joints [-2.843, -70.015, 127.1, -183.79, 56.951, 242.191] to (-316.66, 5.05, -216.79) mm, rotated rx -179.15 ry 0 rz -30.08 deg; joints [-2.846, -70.007, 127.102, -183.793, 56.961, 242.192]
  MoveL 4934 to (-316.66, 5.05, -216.79) mm, rotated rx -179.15 ry 0 rz -30.08 deg; joints [-2.846, -70.007, 127.102, -183.793, 56.961, 242.192]
  MoveL 4935 to (-327.16, -13.08, -216.79) mm, rotated rx -179.15 ry 0 rz -30.08 deg; joints [-3.341, -68.976, 127.38, -184.32, 58.286, 242.394]
  MoveC 4936 to (-327.25, -13.19, -216.79) mm, rotated rx -179.15 ry 0 rz -30.08 deg; joints [-3.345, -68.969, 127.381, -184.324, 58.294, 242.396] to (-327.36, -13.29, -216.79) mm, rotated rx -179.15 ry 0 rz -30.08 deg; joints [-3.35, -68.963, 127.383, -184.33, 58.301, 242.399]
  MoveL 4937 to (-327.36, -13.29, -216.79) mm, rotated rx -179.15 ry 0 rz -30.08 deg; joints [-3.35, -68.963, 127.383, -184.33, 58.301, 242.399]
  MoveC 4938 to (-327.47, -13.38, -216.79) mm, rotated rx -179.15 ry 0 rz -30.08 deg; joints [-3.355, -68.958, 127.384, -184.336, 58.308, 242.401] to (-327.55, -13.5, -216.79) mm, rotated rx -179.15 ry 0 rz -30.08 deg; joints [-3.359, -68.951, 127.385, -184.34, 58.316, 242.403]
  MoveL 4939 to (-327.55, -13.5, -216.79) mm, rotated rx -179.15 ry 0 rz -30.08 deg; joints [-3.359, -68.951, 127.385, -184.34, 58.316, 242.403]
  MoveC 4940 to (-328.23, -14.66, -217.35) mm, rotated rx -179.15 ry 0 rz -30.08 deg; joints [-3.39, -68.855, 127.358, -184.372, 58.386, 242.416] to (-328.51, -15.14, -218.69) mm, rotated rx -179.15 ry 0 rz -30.08 deg; joints [-3.399, -68.758, 127.26, -184.384, 58.385, 242.422]
  MoveL 4941 to (-328.51, -15.14, -218.69) mm, rotated rx -179.15 ry 0 rz -30.08 deg; joints [-3.399, -68.758, 127.26, -184.384, 58.385, 242.422]
  MoveL 4942 to (-328.51, -15.14, -221.23) mm, rotated rx -179.15 ry 0 rz -30.08 deg; joints [-3.392, -68.629, 127.062, -184.379, 58.317, 242.423]
  MoveC 4943 to (-328.23, -14.66, -222.58) mm, rotated rx -179.15 ry 0 rz -30.08 deg; joints [-3.375, -68.588, 126.95, -184.362, 58.246, 242.419] to (-327.55, -13.5, -223.14) mm, rotated rx -179.15 ry 0 rz -30.08 deg; joints [-3.342, -68.626, 126.89, -184.328, 58.146, 242.408]
  MoveL 4944 to (-327.55, -13.5, -223.14) mm, rotated rx -179.15 ry 0 rz -30.08 deg; joints [-3.342, -68.626, 126.89, -184.328, 58.146, 242.408]
  MoveC 4945 to (-327.47, -13.38, -223.14) mm, rotated rx -179.15 ry 0 rz -30.08 deg; joints [-3.338, -68.633, 126.889, -184.324, 58.138, 242.406] to (-327.36, -13.29, -223.14) mm, rotated rx -179.15 ry 0 rz -30.08 deg; joints [-3.333, -68.638, 126.888, -184.318, 58.131, 242.403]
  MoveL 4946 to (-327.36, -13.29, -223.14) mm, rotated rx -179.15 ry 0 rz -30.08 deg; joints [-3.333, -68.638, 126.888, -184.318, 58.131, 242.403]
  MoveC 4947 to (-327.25, -13.19, -223.14) mm, rotated rx -179.15 ry 0 rz -30.08 deg; joints [-3.328, -68.644, 126.887, -184.312, 58.124, 242.401] to (-327.16, -13.08, -223.14) mm, rotated rx -179.15 ry 0 rz -30.08 deg; joints [-3.324, -68.651, 126.885, -184.308, 58.116, 242.399]
  MoveL 4948 to (-327.16, -13.08, -223.14) mm, rotated rx -179.15 ry 0 rz -30.08 deg; joints [-3.324, -68.651, 126.885, -184.308, 58.116, 242.399]
  MoveL 4949 to (-316.66, 5.05, -223.14) mm, rotated rx -179.15 ry 0 rz -30.08 deg; joints [-2.831, -69.675, 126.608, -183.782, 56.799, 242.196]
  MoveC 4950 to (-316.6, 5.19, -223.14) mm, rotated rx -179.15 ry 0 rz -30.08 deg; joints [-2.829, -69.682, 126.606, -183.78, 56.79, 242.195] to (-316.58, 5.33, -223.14) mm, rotated rx -179.15 ry 0 rz -30.08 deg; joints [-2.828, -69.69, 126.604, -183.779, 56.779, 242.195]
  MoveL 4951 to (-316.58, 5.33, -223.14) mm, rotated rx -179.15 ry 0 rz -30.08 deg; joints [-2.828, -69.69, 126.604, -183.779, 56.779, 242.195]
  MoveC 4952 to (-316.55, 5.47, -223.14) mm, rotated rx -179.15 ry 0 rz -30.08 deg; joints [-2.826, -69.698, 126.601, -183.778, 56.769, 242.195] to (-316.49, 5.6, -223.14) mm, rotated rx -179.15 ry 0 rz -30.08 deg; joints [-2.824, -69.705, 126.599, -183.775, 56.76, 242.194]
  MoveL 4953 to (-316.49, 5.6, -223.14) mm, rotated rx -179.15 ry 0 rz -30.08 deg; joints [-2.824, -69.705, 126.599, -183.775, 56.76, 242.194]
  MoveC 4954 to (-315.82, 6.77, -223.69) mm, rotated rx -179.15 ry 0 rz -30.08 deg; joints [-2.791, -69.741, 126.536, -183.74, 56.66, 242.18] to (-315.54, 7.25, -225.04) mm, rotated rx -179.15 ry 0 rz -30.08 deg; joints [-2.775, -69.697, 126.424, -183.723, 56.591, 242.175]
  MoveL 4955 to (-315.54, 7.25, -225.04) mm, rotated rx -179.15 ry 0 rz -30.08 deg; joints [-2.775, -69.697, 126.424, -183.723, 56.591, 242.175]
  MoveL 4956 to (-315.54, 7.25, -227.58) mm, rotated rx -179.15 ry 0 rz -30.08 deg; joints [-2.769, -69.564, 126.226, -183.72, 56.526, 242.176]
  MoveC 4957 to (-315.82, 6.77, -228.93) mm, rotated rx -179.15 ry 0 rz -30.08 deg; joints [-2.779, -69.466, 126.129, -183.732, 56.527, 242.183] to (-316.49, 5.6, -229.49) mm, rotated rx -179.15 ry 0 rz -30.08 deg; joints [-2.809, -69.373, 126.104, -183.765, 56.597, 242.197]
  MoveL 4958 to (-316.49, 5.6, -229.49) mm, rotated rx -179.15 ry 0 rz -30.08 deg; joints [-2.809, -69.373, 126.104, -183.765, 56.597, 242.197]
  MoveC 4959 to (-316.55, 5.47, -229.49) mm, rotated rx -179.15 ry 0 rz -30.08 deg; joints [-2.812, -69.366, 126.106, -183.768, 56.606, 242.198] to (-316.58, 5.33, -229.49) mm, rotated rx -179.15 ry 0 rz -30.08 deg; joints [-2.813, -69.358, 126.109, -183.769, 56.616, 242.198]
  MoveL 4960 to (-316.58, 5.33, -229.49) mm, rotated rx -179.15 ry 0 rz -30.08 deg; joints [-2.813, -69.358, 126.109, -183.769, 56.616, 242.198]
  MoveC 4961 to (-316.6, 5.18, -229.49) mm, rotated rx -179.15 ry 0 rz -30.08 deg; joints [-2.815, -69.35, 126.111, -183.77, 56.627, 242.198] to (-316.66, 5.05, -229.49) mm, rotated rx -179.15 ry 0 rz -30.08 deg; joints [-2.817, -69.343, 126.113, -183.773, 56.636, 242.199]
  MoveL 4962 to (-316.66, 5.05, -229.49) mm, rotated rx -179.15 ry 0 rz -30.08 deg; joints [-2.817, -69.343, 126.113, -183.773, 56.636, 242.199]
  MoveL 4963 to (-327.16, -13.08, -229.49) mm, rotated rx -179.15 ry 0 rz -30.08 deg; joints [-3.307, -68.326, 126.389, -184.296, 57.944, 242.404]
  MoveC 4964 to (-327.25, -13.19, -229.49) mm, rotated rx -179.15 ry 0 rz -30.08 deg; joints [-3.311, -68.319, 126.39, -184.3, 57.952, 242.406] to (-327.36, -13.29, -229.49) mm, rotated rx -179.15 ry 0 rz -30.08 deg; joints [-3.316, -68.314, 126.392, -184.306, 57.959, 242.408]
  MoveL 4965 to (-327.36, -13.29, -229.49) mm, rotated rx -179.15 ry 0 rz -30.08 deg; joints [-3.316, -68.314, 126.392, -184.306, 57.959, 242.408]
  MoveC 4966 to (-327.47, -13.38, -229.49) mm, rotated rx -179.15 ry 0 rz -30.08 deg; joints [-3.321, -68.308, 126.393, -184.312, 57.966, 242.411] to (-327.55, -13.5, -229.49) mm, rotated rx -179.15 ry 0 rz -30.08 deg; joints [-3.325, -68.302, 126.394, -184.316, 57.974, 242.413]
  MoveL 4967 to (-327.55, -13.5, -229.49) mm, rotated rx -179.15 ry 0 rz -30.08 deg; joints [-3.325, -68.301, 126.394, -184.316, 57.974, 242.413]
  MoveC 4968 to (-328.23, -14.66, -230.04) mm, rotated rx -179.15 ry 0 rz -30.08 deg; joints [-3.355, -68.207, 126.367, -184.348, 58.043, 242.425] to (-328.51, -15.14, -231.39) mm, rotated rx -179.15 ry 0 rz -30.08 deg; joints [-3.365, -68.11, 126.268, -184.36, 58.041, 242.431]
  MoveL 4969 to (-328.51, -15.14, -231.39) mm, rotated rx -179.15 ry 0 rz -30.08 deg; joints [-3.365, -68.11, 126.268, -184.36, 58.041, 242.431]
  MoveL 4970 to (-328.51, -15.14, -233.93) mm, rotated rx -179.15 ry 0 rz -30.08 deg; joints [-3.358, -67.981, 126.069, -184.355, 57.971, 242.433]
  MoveC 4971 to (-328.23, -14.66, -235.28) mm, rotated rx -179.15 ry 0 rz -30.08 deg; joints [-3.342, -67.94, 125.957, -184.339, 57.899, 242.429] to (-327.55, -13.5, -235.83) mm, rotated rx -179.15 ry 0 rz -30.08 deg; joints [-3.309, -67.977, 125.896, -184.305, 57.801, 242.418]
  MoveL 4972 to (-327.55, -13.5, -235.83) mm, rotated rx -179.15 ry 0 rz -30.08 deg; joints [-3.309, -67.977, 125.896, -184.305, 57.801, 242.418]
  MoveC 4973 to (-327.47, -13.38, -235.83) mm, rotated rx -179.15 ry 0 rz -30.08 deg; joints [-3.305, -67.984, 125.895, -184.3, 57.792, 242.416] to (-327.36, -13.29, -235.83) mm, rotated rx -179.15 ry 0 rz -30.08 deg; joints [-3.3, -67.989, 125.894, -184.295, 57.786, 242.413]
  MoveL 4974 to (-327.36, -13.29, -235.83) mm, rotated rx -179.15 ry 0 rz -30.08 deg; joints [-3.3, -67.989, 125.894, -184.295, 57.786, 242.413]
  MoveC 4975 to (-327.25, -13.19, -235.83) mm, rotated rx -179.15 ry 0 rz -30.08 deg; joints [-3.294, -67.995, 125.893, -184.289, 57.779, 242.411] to (-327.16, -13.08, -235.83) mm, rotated rx -179.15 ry 0 rz -30.08 deg; joints [-3.29, -68.001, 125.891, -184.284, 57.771, 242.409]
  MoveL 4976 to (-327.16, -13.08, -235.83) mm, rotated rx -179.15 ry 0 rz -30.08 deg; joints [-3.29, -68.001, 125.891, -184.284, 57.771, 242.409]
  MoveL 4977 to (-316.66, 5.05, -235.83) mm, rotated rx -179.15 ry 0 rz -30.08 deg; joints [-2.803, -69.011, 125.617, -183.763, 56.471, 242.203]
  MoveC 4978 to (-316.6, 5.19, -235.83) mm, rotated rx -179.15 ry 0 rz -30.08 deg; joints [-2.8, -69.019, 125.615, -183.76, 56.462, 242.202] to (-316.58, 5.33, -235.83) mm, rotated rx -179.15 ry 0 rz -30.08 deg; joints [-2.799, -69.026, 125.612, -183.759, 56.451, 242.202]
  MoveL 4979 to (-316.58, 5.33, -235.83) mm, rotated rx -179.15 ry 0 rz -30.08 deg; joints [-2.799, -69.026, 125.612, -183.759, 56.451, 242.202]
  MoveC 4980 to (-316.55, 5.47, -235.83) mm, rotated rx -179.15 ry 0 rz -30.08 deg; joints [-2.798, -69.034, 125.61, -183.758, 56.441, 242.202] to (-316.49, 5.6, -235.83) mm, rotated rx -179.15 ry 0 rz -30.08 deg; joints [-2.795, -69.041, 125.608, -183.755, 56.432, 242.201]
  MoveL 4981 to (-316.49, 5.6, -235.83) mm, rotated rx -179.15 ry 0 rz -30.08 deg; joints [-2.795, -69.041, 125.608, -183.755, 56.432, 242.201]
  MoveC 4982 to (-315.82, 6.77, -236.39) mm, rotated rx -179.15 ry 0 rz -30.08 deg; joints [-2.763, -69.076, 125.545, -183.72, 56.333, 242.187] to (-315.54, 7.25, -237.74) mm, rotated rx -179.15 ry 0 rz -30.08 deg; joints [-2.747, -69.032, 125.432, -183.704, 56.264, 242.182]
  MoveL 4983 to (-315.54, 7.25, -237.74) mm, rotated rx -179.15 ry 0 rz -30.08 deg; joints [-2.747, -69.032, 125.432, -183.704, 56.264, 242.182]
  MoveL 4984 to (-315.54, 7.25, -240.28) mm, rotated rx -179.15 ry 0 rz -30.08 deg; joints [-2.741, -68.899, 125.232, -183.701, 56.197, 242.183]
  MoveC 4985 to (-315.82, 6.77, -241.63) mm, rotated rx -179.15 ry 0 rz -30.08 deg; joints [-2.751, -68.802, 125.135, -183.713, 56.196, 242.19] to (-316.49, 5.6, -242.18) mm, rotated rx -179.15 ry 0 rz -30.08 deg; joints [-2.781, -68.71, 125.11, -183.746, 56.265, 242.205]
  MoveL 4986 to (-316.49, 5.6, -242.18) mm, rotated rx -179.15 ry 0 rz -30.08 deg; joints [-2.781, -68.71, 125.11, -183.746, 56.265, 242.205]
  MoveC 4987 to (-316.55, 5.47, -242.18) mm, rotated rx -179.15 ry 0 rz -30.08 deg; joints [-2.784, -68.703, 125.112, -183.749, 56.274, 242.206] to (-316.58, 5.33, -242.18) mm, rotated rx -179.15 ry 0 rz -30.08 deg; joints [-2.785, -68.695, 125.114, -183.75, 56.285, 242.206]
  MoveL 4988 to (-316.58, 5.33, -242.18) mm, rotated rx -179.15 ry 0 rz -30.08 deg; joints [-2.785, -68.695, 125.114, -183.75, 56.285, 242.206]
  MoveC 4989 to (-316.6, 5.18, -242.18) mm, rotated rx -179.15 ry 0 rz -30.08 deg; joints [-2.787, -68.687, 125.117, -183.751, 56.295, 242.206] to (-316.66, 5.05, -242.18) mm, rotated rx -179.15 ry 0 rz -30.08 deg; joints [-2.789, -68.68, 125.119, -183.753, 56.304, 242.207]
  MoveL 4990 to (-316.66, 5.05, -242.18) mm, rotated rx -179.15 ry 0 rz -30.08 deg; joints [-2.789, -68.68, 125.119, -183.753, 56.304, 242.207]
  MoveL 4991 to (-327.16, -13.08, -242.18) mm, rotated rx -179.15 ry 0 rz -30.08 deg; joints [-3.274, -67.677, 125.392, -184.273, 57.595, 242.414]
  MoveC 4992 to (-327.25, -13.19, -242.18) mm, rotated rx -179.15 ry 0 rz -30.08 deg; joints [-3.278, -67.671, 125.393, -184.278, 57.604, 242.416] to (-327.36, -13.29, -242.18) mm, rotated rx -179.15 ry 0 rz -30.08 deg; joints [-3.283, -67.665, 125.395, -184.283, 57.61, 242.418]
  MoveL 4993 to (-327.36, -13.29, -242.18) mm, rotated rx -179.15 ry 0 rz -30.08 deg; joints [-3.283, -67.665, 125.395, -184.283, 57.61, 242.418]
  MoveC 4994 to (-327.47, -13.38, -242.18) mm, rotated rx -179.15 ry 0 rz -30.08 deg; joints [-3.288, -67.66, 125.396, -184.289, 57.617, 242.421] to (-327.55, -13.5, -242.18) mm, rotated rx -179.15 ry 0 rz -30.08 deg; joints [-3.292, -67.653, 125.397, -184.293, 57.625, 242.423]
  MoveL 4995 to (-327.55, -13.5, -242.18) mm, rotated rx -179.15 ry 0 rz -30.08 deg; joints [-3.292, -67.653, 125.397, -184.293, 57.625, 242.423]
  MoveC 4996 to (-328.23, -14.66, -242.74) mm, rotated rx -179.15 ry 0 rz -30.08 deg; joints [-3.322, -67.559, 125.369, -184.325, 57.692, 242.436] to (-328.51, -15.14, -244.09) mm, rotated rx -179.15 ry 0 rz -30.08 deg; joints [-3.331, -67.464, 125.27, -184.337, 57.689, 242.442]
  MoveL 4997 to (-328.51, -15.14, -244.09) mm, rotated rx -179.15 ry 0 rz -30.08 deg; joints [-3.331, -67.464, 125.27, -184.337, 57.689, 242.442]
  MoveL 4998 to (-328.51, -15.14, -246.63) mm, rotated rx -179.15 ry 0 rz -30.08 deg; joints [-3.325, -67.335, 125.07, -184.332, 57.618, 242.444]
  MoveC 4999 to (-328.23, -14.66, -247.97) mm, rotated rx -179.15 ry 0 rz -30.08 deg; joints [-3.308, -67.293, 124.957, -184.316, 57.546, 242.44] to (-327.55, -13.5, -248.53) mm, rotated rx -179.15 ry 0 rz -30.08 deg; joints [-3.276, -67.33, 124.896, -184.282, 57.448, 242.428]
  MoveL 5000 to (-327.55, -13.5, -248.53) mm, rotated rx -179.15 ry 0 rz -30.08 deg; joints [-3.276, -67.33, 124.896, -184.282, 57.448, 242.428]
  MoveC 5001 to (-327.47, -13.38, -248.53) mm, rotated rx -179.15 ry 0 rz -30.08 deg; joints [-3.272, -67.336, 124.895, -184.278, 57.44, 242.426] to (-327.36, -13.29, -248.53) mm, rotated rx -179.15 ry 0 rz -30.08 deg; joints [-3.267, -67.341, 124.894, -184.272, 57.433, 242.424]
  MoveL 5002 to (-327.36, -13.29, -248.53) mm, rotated rx -179.15 ry 0 rz -30.08 deg; joints [-3.267, -67.341, 124.894, -184.272, 57.433, 242.424]
  MoveC 5003 to (-327.25, -13.19, -248.53) mm, rotated rx -179.15 ry 0 rz -30.08 deg; joints [-3.262, -67.347, 124.893, -184.267, 57.426, 242.421] to (-327.16, -13.08, -248.53) mm, rotated rx -179.15 ry 0 rz -30.08 deg; joints [-3.258, -67.353, 124.891, -184.262, 57.418, 242.419]
  MoveL 5004 to (-327.16, -13.08, -248.53) mm, rotated rx -179.15 ry 0 rz -30.08 deg; joints [-3.258, -67.353, 124.891, -184.262, 57.418, 242.419]
  MoveL 5005 to (-316.66, 5.05, -248.53) mm, rotated rx -179.15 ry 0 rz -30.08 deg; joints [-2.775, -68.349, 124.619, -183.744, 56.135, 242.211]
  MoveC 5006 to (-316.6, 5.19, -248.53) mm, rotated rx -179.15 ry 0 rz -30.08 deg; joints [-2.773, -68.356, 124.617, -183.741, 56.126, 242.21] to (-316.58, 5.33, -248.53) mm, rotated rx -179.15 ry 0 rz -30.08 deg; joints [-2.772, -68.364, 124.615, -183.74, 56.116, 242.21]
  MoveL 5007 to (-316.58, 5.33, -248.53) mm, rotated rx -179.15 ry 0 rz -30.08 deg; joints [-2.772, -68.364, 124.615, -183.74, 56.116, 242.21]
  MoveC 5008 to (-316.55, 5.47, -248.53) mm, rotated rx -179.15 ry 0 rz -30.08 deg; joints [-2.77, -68.372, 124.612, -183.739, 56.106, 242.21] to (-316.49, 5.6, -248.53) mm, rotated rx -179.15 ry 0 rz -30.08 deg; joints [-2.768, -68.379, 124.61, -183.737, 56.096, 242.209]
  MoveL 5009 to (-316.49, 5.6, -248.53) mm, rotated rx -179.15 ry 0 rz -30.08 deg; joints [-2.768, -68.379, 124.61, -183.737, 56.096, 242.209]
  MoveC 5010 to (-315.82, 6.77, -249.09) mm, rotated rx -179.15 ry 0 rz -30.08 deg; joints [-2.735, -68.413, 124.547, -183.702, 55.999, 242.195] to (-315.54, 7.25, -250.44) mm, rotated rx -179.15 ry 0 rz -30.08 deg; joints [-2.72, -68.368, 124.433, -183.686, 55.928, 242.19]
  MoveL 5011 to (-315.54, 7.25, -250.44) mm, rotated rx -179.15 ry 0 rz -30.08 deg; joints [-2.72, -68.368, 124.433, -183.686, 55.928, 242.19]
  MoveL 5012 to (-315.54, 7.25, -252.98) mm, rotated rx -179.15 ry 0 rz -30.08 deg; joints [-2.714, -68.236, 124.233, -183.683, 55.861, 242.191]
  MoveC 5013 to (-315.82, 6.77, -254.32) mm, rotated rx -179.15 ry 0 rz -30.08 deg; joints [-2.724, -68.14, 124.134, -183.695, 55.858, 242.198] to (-316.49, 5.6, -254.88) mm, rotated rx -179.15 ry 0 rz -30.08 deg; joints [-2.754, -68.048, 124.109, -183.728, 55.926, 242.213]
  MoveL 5014 to (-316.49, 5.6, -254.88) mm, rotated rx -179.15 ry 0 rz -30.08 deg; joints [-2.754, -68.048, 124.109, -183.728, 55.926, 242.213]
  MoveC 5015 to (-316.55, 5.47, -254.88) mm, rotated rx -179.15 ry 0 rz -30.08 deg; joints [-2.757, -68.041, 124.111, -183.73, 55.935, 242.214] to (-316.58, 5.33, -254.88) mm, rotated rx -179.15 ry 0 rz -30.08 deg; joints [-2.758, -68.033, 124.113, -183.731, 55.945, 242.214]
  MoveL 5016 to (-316.58, 5.33, -254.88) mm, rotated rx -179.15 ry 0 rz -30.08 deg; joints [-2.758, -68.033, 124.113, -183.731, 55.945, 242.214]
  MoveC 5017 to (-316.6, 5.18, -254.88) mm, rotated rx -179.15 ry 0 rz -30.08 deg; joints [-2.759, -68.026, 124.116, -183.732, 55.955, 242.214] to (-316.66, 5.05, -254.88) mm, rotated rx -179.15 ry 0 rz -30.08 deg; joints [-2.762, -68.019, 124.118, -183.735, 55.964, 242.215]
  MoveL 5018 to (-316.66, 5.05, -254.88) mm, rotated rx -179.15 ry 0 rz -30.08 deg; joints [-2.762, -68.019, 124.118, -183.735, 55.964, 242.215]
  MoveL 5019 to (-327.16, -13.08, -254.88) mm, rotated rx -179.15 ry 0 rz -30.08 deg; joints [-3.242, -67.03, 124.389, -184.252, 57.239, 242.425]
  MoveC 5020 to (-327.25, -13.19, -254.88) mm, rotated rx -179.15 ry 0 rz -30.08 deg; joints [-3.246, -67.023, 124.39, -184.256, 57.248, 242.426] to (-327.36, -13.29, -254.88) mm, rotated rx -179.15 ry 0 rz -30.08 deg; joints [-3.251, -67.018, 124.391, -184.262, 57.254, 242.429]
  MoveL 5021 to (-327.36, -13.29, -254.88) mm, rotated rx -179.15 ry 0 rz -30.08 deg; joints [-3.251, -67.018, 124.391, -184.262, 57.254, 242.429]
  MoveC 5022 to (-327.47, -13.38, -254.88) mm, rotated rx -179.15 ry 0 rz -30.08 deg; joints [-3.256, -67.013, 124.392, -184.267, 57.261, 242.432] to (-327.55, -13.5, -254.88) mm, rotated rx -179.15 ry 0 rz -30.08 deg; joints [-3.26, -67.006, 124.394, -184.272, 57.269, 242.434]
  MoveL 5023 to (-327.55, -13.5, -254.88) mm, rotated rx -179.15 ry 0 rz -30.08 deg; joints [-3.26, -67.006, 124.394, -184.272, 57.269, 242.434]
  MoveC 5024 to (-328.23, -14.66, -255.44) mm, rotated rx -179.15 ry 0 rz -30.08 deg; joints [-3.289, -66.913, 124.366, -184.304, 57.335, 242.447] to (-328.51, -15.14, -256.79) mm, rotated rx -179.15 ry 0 rz -30.08 deg; joints [-3.298, -66.818, 124.266, -184.315, 57.33, 242.453]
  MoveL 5025 to (-328.51, -15.14, -256.79) mm, rotated rx -179.15 ry 0 rz -30.08 deg; joints [-3.298, -66.818, 124.266, -184.315, 57.33, 242.453]
  MoveL 5026 to (-328.51, -15.14, -259.32) mm, rotated rx -179.15 ry 0 rz -30.08 deg; joints [-3.292, -66.689, 124.064, -184.311, 57.257, 242.455]
  MoveC 5027 to (-328.23, -14.66, -260.67) mm, rotated rx -179.15 ry 0 rz -30.08 deg; joints [-3.276, -66.647, 123.95, -184.295, 57.185, 242.451] to (-327.55, -13.5, -261.23) mm, rotated rx -179.15 ry 0 rz -30.08 deg; joints [-3.244, -66.683, 123.89, -184.261, 57.088, 242.439]
  MoveL 5028 to (-327.55, -13.5, -261.23) mm, rotated rx -179.15 ry 0 rz -30.08 deg; joints [-3.244, -66.683, 123.89, -184.261, 57.088, 242.439]
  MoveC 5029 to (-327.47, -13.38, -261.23) mm, rotated rx -179.15 ry 0 rz -30.08 deg; joints [-3.24, -66.689, 123.888, -184.257, 57.08, 242.437] to (-327.36, -13.29, -261.23) mm, rotated rx -179.15 ry 0 rz -30.08 deg; joints [-3.235, -66.695, 123.887, -184.251, 57.073, 242.435]
  MoveL 5030 to (-327.36, -13.29, -261.23) mm, rotated rx -179.15 ry 0 rz -30.08 deg; joints [-3.235, -66.695, 123.887, -184.251, 57.073, 242.435]
  MoveC 5031 to (-327.25, -13.19, -261.23) mm, rotated rx -179.15 ry 0 rz -30.08 deg; joints [-3.23, -66.7, 123.886, -184.246, 57.067, 242.432] to (-327.16, -13.08, -261.23) mm, rotated rx -179.15 ry 0 rz -30.08 deg; joints [-3.226, -66.706, 123.885, -184.241, 57.059, 242.43]
  MoveL 5032 to (-327.16, -13.08, -261.23) mm, rotated rx -179.15 ry 0 rz -30.08 deg; joints [-3.226, -66.706, 123.885, -184.241, 57.059, 242.43]
  MoveL 5033 to (-316.66, 5.05, -261.23) mm, rotated rx -179.15 ry 0 rz -30.08 deg; joints [-2.748, -67.689, 123.615, -183.726, 55.792, 242.22]
  MoveC 5034 to (-316.6, 5.19, -261.23) mm, rotated rx -179.15 ry 0 rz -30.08 deg; joints [-2.746, -67.696, 123.613, -183.724, 55.782, 242.219] to (-316.58, 5.33, -261.23) mm, rotated rx -179.15 ry 0 rz -30.08 deg; joints [-2.744, -67.703, 123.611, -183.723, 55.772, 242.219]
  MoveL 5035 to (-316.58, 5.33, -261.23) mm, rotated rx -179.15 ry 0 rz -30.08 deg; joints [-2.744, -67.703, 123.611, -183.723, 55.772, 242.219]
  MoveC 5036 to (-316.55, 5.47, -261.23) mm, rotated rx -179.15 ry 0 rz -30.08 deg; joints [-2.743, -67.711, 123.608, -183.722, 55.762, 242.218] to (-316.49, 5.6, -261.23) mm, rotated rx -179.15 ry 0 rz -30.08 deg; joints [-2.741, -67.718, 123.606, -183.719, 55.753, 242.217]
  MoveL 5037 to (-316.49, 5.6, -261.23) mm, rotated rx -179.15 ry 0 rz -30.08 deg; joints [-2.741, -67.718, 123.606, -183.719, 55.753, 242.217]
  MoveC 5038 to (-315.82, 6.77, -261.79) mm, rotated rx -179.15 ry 0 rz -30.08 deg; joints [-2.709, -67.751, 123.543, -183.685, 55.656, 242.203] to (-315.54, 7.25, -263.13) mm, rotated rx -179.15 ry 0 rz -30.08 deg; joints [-2.693, -67.706, 123.429, -183.669, 55.586, 242.198]
  MoveL 5039 to (-315.54, 7.25, -263.13) mm, rotated rx -179.15 ry 0 rz -30.08 deg; joints [-2.693, -67.706, 123.429, -183.669, 55.586, 242.198]
  MoveL 5040 to (-315.54, 7.25, -265.67) mm, rotated rx -179.15 ry 0 rz -30.08 deg; joints [-2.688, -67.574, 123.227, -183.666, 55.516, 242.2]
  MoveC 5041 to (-315.82, 6.77, -267.02) mm, rotated rx -179.15 ry 0 rz -30.08 deg; joints [-2.698, -67.478, 123.128, -183.678, 55.513, 242.207] to (-316.49, 5.6, -267.58) mm, rotated rx -179.15 ry 0 rz -30.08 deg; joints [-2.727, -67.388, 123.102, -183.71, 55.579, 242.222]
  MoveL 5042 to (-316.49, 5.6, -267.58) mm, rotated rx -179.15 ry 0 rz -30.08 deg; joints [-2.727, -67.388, 123.102, -183.71, 55.579, 242.222]
  MoveC 5043 to (-316.55, 5.47, -267.58) mm, rotated rx -179.15 ry 0 rz -30.08 deg; joints [-2.73, -67.381, 123.104, -183.713, 55.588, 242.223] to (-316.58, 5.33, -267.58) mm, rotated rx -179.15 ry 0 rz -30.08 deg; joints [-2.731, -67.373, 123.106, -183.714, 55.598, 242.223]
  MoveL 5044 to (-316.58, 5.33, -267.58) mm, rotated rx -179.15 ry 0 rz -30.08 deg; joints [-2.731, -67.373, 123.106, -183.714, 55.598, 242.223]
  MoveC 5045 to (-316.6, 5.18, -267.58) mm, rotated rx -179.15 ry 0 rz -30.08 deg; joints [-2.732, -67.366, 123.109, -183.715, 55.608, 242.223] to (-316.66, 5.05, -267.58) mm, rotated rx -179.15 ry 0 rz -30.08 deg; joints [-2.735, -67.359, 123.111, -183.718, 55.617, 242.224]
  MoveL 5046 to (-316.66, 5.05, -267.58) mm, rotated rx -179.15 ry 0 rz -30.08 deg; joints [-2.735, -67.359, 123.111, -183.718, 55.617, 242.224]
  MoveL 5047 to (-327.16, -13.08, -267.58) mm, rotated rx -179.15 ry 0 rz -30.08 deg; joints [-3.21, -66.383, 123.379, -184.231, 56.876, 242.436]
  MoveC 5048 to (-327.25, -13.19, -267.58) mm, rotated rx -179.15 ry 0 rz -30.08 deg; joints [-3.214, -66.377, 123.381, -184.236, 56.884, 242.438] to (-327.36, -13.29, -267.58) mm, rotated rx -179.15 ry 0 rz -30.08 deg; joints [-3.219, -66.372, 123.382, -184.241, 56.891, 242.441]
  MoveL 5049 to (-327.36, -13.29, -267.58) mm, rotated rx -179.15 ry 0 rz -30.08 deg; joints [-3.219, -66.372, 123.382, -184.241, 56.891, 242.441]
  MoveC 5050 to (-327.47, -13.38, -267.58) mm, rotated rx -179.15 ry 0 rz -30.08 deg; joints [-3.224, -66.366, 123.383, -184.247, 56.897, 242.443] to (-327.55, -13.5, -267.58) mm, rotated rx -179.15 ry 0 rz -30.08 deg; joints [-3.228, -66.36, 123.384, -184.251, 56.905, 242.445]
  MoveL 5051 to (-327.55, -13.5, -267.58) mm, rotated rx -179.15 ry 0 rz -30.08 deg; joints [-3.228, -66.36, 123.384, -184.251, 56.905, 242.445]
  MoveC 5052 to (-328.23, -14.66, -268.14) mm, rotated rx -179.15 ry 0 rz -30.08 deg; joints [-3.257, -66.268, 123.356, -184.283, 56.97, 242.458] to (-328.51, -15.14, -269.48) mm, rotated rx -179.15 ry 0 rz -30.08 deg; joints [-3.266, -66.173, 123.255, -184.294, 56.964, 242.465]
  MoveL 5053 to (-328.51, -15.14, -269.48) mm, rotated rx -179.15 ry 0 rz -30.08 deg; joints [-3.266, -66.173, 123.255, -184.294, 56.964, 242.465]
  MoveL 5054 to (-328.51, -15.14, -272.02) mm, rotated rx -179.15 ry 0 rz -30.08 deg; joints [-3.26, -66.044, 123.052, -184.29, 56.89, 242.467]
  MoveC 5055 to (-328.23, -14.66, -273.37) mm, rotated rx -179.15 ry 0 rz -30.08 deg; joints [-3.244, -66.002, 122.938, -184.275, 56.817, 242.463] to (-327.55, -13.5, -273.93) mm, rotated rx -179.15 ry 0 rz -30.08 deg; joints [-3.212, -66.037, 122.877, -184.241, 56.721, 242.451]
  MoveL 5056 to (-327.55, -13.5, -273.93) mm, rotated rx -179.15 ry 0 rz -30.08 deg; joints [-3.212, -66.037, 122.877, -184.241, 56.721, 242.451]
  MoveC 5057 to (-327.47, -13.38, -273.93) mm, rotated rx -179.15 ry 0 rz -30.08 deg; joints [-3.208, -66.043, 122.876, -184.237, 56.713, 242.449] to (-327.36, -13.29, -273.93) mm, rotated rx -179.15 ry 0 rz -30.08 deg; joints [-3.203, -66.049, 122.875, -184.231, 56.706, 242.447]
  MoveL 5058 to (-327.36, -13.29, -273.93) mm, rotated rx -179.15 ry 0 rz -30.08 deg; joints [-3.203, -66.049, 122.875, -184.231, 56.706, 242.447]
  MoveC 5059 to (-327.25, -13.19, -273.93) mm, rotated rx -179.15 ry 0 rz -30.08 deg; joints [-3.198, -66.054, 122.874, -184.226, 56.7, 242.444] to (-327.16, -13.08, -273.93) mm, rotated rx -179.15 ry 0 rz -30.08 deg; joints [-3.194, -66.06, 122.872, -184.222, 56.692, 242.442]
  MoveL 5060 to (-327.16, -13.08, -273.93) mm, rotated rx -179.15 ry 0 rz -30.08 deg; joints [-3.194, -66.06, 122.872, -184.222, 56.692, 242.442]
  MoveL 5061 to (-316.66, 5.05, -273.93) mm, rotated rx -179.15 ry 0 rz -30.08 deg; joints [-2.722, -67.029, 122.605, -183.71, 55.44, 242.229]
  MoveC 5062 to (-316.6, 5.19, -273.93) mm, rotated rx -179.15 ry 0 rz -30.08 deg; joints [-2.719, -67.036, 122.603, -183.707, 55.431, 242.228] to (-316.58, 5.33, -273.93) mm, rotated rx -179.15 ry 0 rz -30.08 deg; joints [-2.718, -67.043, 122.6, -183.706, 55.421, 242.228]
  MoveL 5063 to (-316.58, 5.33, -273.93) mm, rotated rx -179.15 ry 0 rz -30.08 deg; joints [-2.718, -67.043, 122.6, -183.706, 55.421, 242.228]
  MoveC 5064 to (-316.55, 5.47, -273.93) mm, rotated rx -179.15 ry 0 rz -30.08 deg; joints [-2.717, -67.051, 122.598, -183.705, 55.412, 242.228] to (-316.49, 5.6, -273.93) mm, rotated rx -179.15 ry 0 rz -30.08 deg; joints [-2.714, -67.058, 122.596, -183.702, 55.403, 242.227]
  MoveL 5065 to (-316.49, 5.6, -273.93) mm, rotated rx -179.15 ry 0 rz -30.08 deg; joints [-2.714, -67.058, 122.596, -183.702, 55.403, 242.227]
  MoveC 5066 to (-315.82, 6.77, -274.48) mm, rotated rx -179.15 ry 0 rz -30.08 deg; joints [-2.682, -67.09, 122.533, -183.668, 55.306, 242.213] to (-315.54, 7.25, -275.83) mm, rotated rx -179.15 ry 0 rz -30.08 deg; joints [-2.667, -67.045, 122.417, -183.653, 55.235, 242.208]
  MoveL 5067 to (-315.54, 7.25, -275.83) mm, rotated rx -179.15 ry 0 rz -30.08 deg; joints [-2.667, -67.045, 122.417, -183.653, 55.235, 242.208]
  MoveL 5068 to (-315.54, 7.25, -278.37) mm, rotated rx -179.15 ry 0 rz -30.08 deg; joints [-2.662, -66.913, 122.214, -183.65, 55.164, 242.209]
  MoveC 5069 to (-315.82, 6.77, -279.72) mm, rotated rx -179.15 ry 0 rz -30.08 deg; joints [-2.672, -66.818, 122.114, -183.662, 55.16, 242.217] to (-316.49, 5.6, -280.28) mm, rotated rx -179.15 ry 0 rz -30.08 deg; joints [-2.701, -66.728, 122.088, -183.694, 55.224, 242.232]
  MoveL 5070 to (-316.49, 5.6, -280.28) mm, rotated rx -179.15 ry 0 rz -30.08 deg; joints [-2.701, -66.728, 122.088, -183.694, 55.224, 242.232]
  MoveC 5071 to (-316.55, 5.47, -280.28) mm, rotated rx -179.15 ry 0 rz -30.08 deg; joints [-2.703, -66.721, 122.09, -183.697, 55.233, 242.233] to (-316.58, 5.33, -280.28) mm, rotated rx -179.15 ry 0 rz -30.08 deg; joints [-2.705, -66.714, 122.093, -183.698, 55.243, 242.233]
  MoveL 5072 to (-316.58, 5.33, -280.28) mm, rotated rx -179.15 ry 0 rz -30.08 deg; joints [-2.705, -66.714, 122.093, -183.698, 55.243, 242.233]
  MoveC 5073 to (-316.6, 5.18, -280.28) mm, rotated rx -179.15 ry 0 rz -30.08 deg; joints [-2.706, -66.707, 122.095, -183.699, 55.253, 242.233] to (-316.66, 5.05, -280.28) mm, rotated rx -179.15 ry 0 rz -30.08 deg; joints [-2.708, -66.7, 122.097, -183.702, 55.262, 242.234]
  MoveL 5074 to (-316.66, 5.05, -280.28) mm, rotated rx -179.15 ry 0 rz -30.08 deg; joints [-2.708, -66.7, 122.097, -183.702, 55.262, 242.234]
  MoveL 5075 to (-327.16, -13.08, -280.28) mm, rotated rx -179.15 ry 0 rz -30.08 deg; joints [-3.179, -65.737, 122.363, -184.212, 56.506, 242.448]
  MoveC 5076 to (-327.25, -13.19, -280.28) mm, rotated rx -179.15 ry 0 rz -30.08 deg; joints [-3.183, -65.731, 122.365, -184.216, 56.514, 242.45] to (-327.36, -13.29, -280.28) mm, rotated rx -179.15 ry 0 rz -30.08 deg; joints [-3.188, -65.726, 122.366, -184.222, 56.52, 242.453]
  MoveL 5077 to (-327.36, -13.29, -280.28) mm, rotated rx -179.15 ry 0 rz -30.08 deg; joints [-3.188, -65.726, 122.366, -184.222, 56.52, 242.453]
  MoveC 5078 to (-327.47, -13.38, -280.28) mm, rotated rx -179.15 ry 0 rz -30.08 deg; joints [-3.193, -65.721, 122.367, -184.228, 56.527, 242.456] to (-327.55, -13.5, -280.28) mm, rotated rx -179.15 ry 0 rz -30.08 deg; joints [-3.196, -65.714, 122.368, -184.232, 56.535, 242.458]
  MoveL 5079 to (-327.55, -13.5, -280.28) mm, rotated rx -179.15 ry 0 rz -30.08 deg; joints [-3.196, -65.714, 122.368, -184.232, 56.535, 242.458]
  MoveC 5080 to (-328.23, -14.66, -280.83) mm, rotated rx -179.15 ry 0 rz -30.08 deg; joints [-3.225, -65.623, 122.34, -184.263, 56.598, 242.471] to (-328.51, -15.14, -282.18) mm, rotated rx -179.15 ry 0 rz -30.08 deg; joints [-3.234, -65.529, 122.238, -184.275, 56.591, 242.478]
  MoveL 5081 to (-328.51, -15.14, -282.18) mm, rotated rx -179.15 ry 0 rz -30.08 deg; joints [-3.234, -65.529, 122.238, -184.275, 56.591, 242.478]
  MoveL 5082 to (-328.51, -15.14, -284.72) mm, rotated rx -179.15 ry 0 rz -30.08 deg; joints [-3.228, -65.4, 122.034, -184.271, 56.515, 242.48]
  MoveC 5083 to (-328.23, -14.66, -286.07) mm, rotated rx -179.15 ry 0 rz -30.08 deg; joints [-3.212, -65.358, 121.919, -184.256, 56.443, 242.476] to (-327.55, -13.5, -286.62) mm, rotated rx -179.15 ry 0 rz -30.08 deg; joints [-3.181, -65.392, 121.858, -184.222, 56.347, 242.464]
  MoveL 5084 to (-327.55, -13.5, -286.62) mm, rotated rx -179.15 ry 0 rz -30.08 deg; joints [-3.181, -65.392, 121.858, -184.222, 56.347, 242.464]
  MoveC 5085 to (-327.47, -13.38, -286.62) mm, rotated rx -179.15 ry 0 rz -30.08 deg; joints [-3.177, -65.398, 121.857, -184.218, 56.339, 242.462] to (-327.36, -13.29, -286.62) mm, rotated rx -179.15 ry 0 rz -30.08 deg; joints [-3.172, -65.403, 121.855, -184.213, 56.333, 242.459]
  MoveL 5086 to (-327.36, -13.29, -286.62) mm, rotated rx -179.15 ry 0 rz -30.08 deg; joints [-3.172, -65.403, 121.855, -184.213, 56.333, 242.459]
  MoveC 5087 to (-327.25, -13.19, -286.62) mm, rotated rx -179.15 ry 0 rz -30.08 deg; joints [-3.167, -65.408, 121.854, -184.207, 56.326, 242.457] to (-327.16, -13.08, -286.62) mm, rotated rx -179.15 ry 0 rz -30.08 deg; joints [-3.163, -65.414, 121.853, -184.203, 56.318, 242.455]
  MoveL 5088 to (-327.16, -13.08, -286.62) mm, rotated rx -179.15 ry 0 rz -30.08 deg; joints [-3.163, -65.414, 121.853, -184.203, 56.318, 242.455]
  MoveL 5089 to (-316.66, 5.05, -286.62) mm, rotated rx -179.15 ry 0 rz -30.08 deg; joints [-2.695, -66.37, 121.588, -183.694, 55.082, 242.239]
  MoveC 5090 to (-316.6, 5.19, -286.62) mm, rotated rx -179.15 ry 0 rz -30.08 deg; joints [-2.693, -66.377, 121.586, -183.691, 55.073, 242.238] to (-316.58, 5.33, -286.62) mm, rotated rx -179.15 ry 0 rz -30.08 deg; joints [-2.692, -66.384, 121.583, -183.69, 55.063, 242.238]
  MoveL 5091 to (-316.58, 5.33, -286.62) mm, rotated rx -179.15 ry 0 rz -30.08 deg; joints [-2.692, -66.384, 121.583, -183.69, 55.063, 242.238]
  MoveC 5092 to (-316.55, 5.47, -286.62) mm, rotated rx -179.15 ry 0 rz -30.08 deg; joints [-2.691, -66.392, 121.581, -183.689, 55.053, 242.238] to (-316.49, 5.6, -286.62) mm, rotated rx -179.15 ry 0 rz -30.08 deg; joints [-2.688, -66.399, 121.579, -183.687, 55.044, 242.237]
  MoveL 5093 to (-316.49, 5.6, -286.62) mm, rotated rx -179.15 ry 0 rz -30.08 deg; joints [-2.688, -66.399, 121.579, -183.687, 55.044, 242.237]
  MoveC 5094 to (-315.82, 6.77, -287.18) mm, rotated rx -179.15 ry 0 rz -30.08 deg; joints [-2.657, -66.43, 121.515, -183.653, 54.949, 242.223] to (-315.54, 7.25, -288.53) mm, rotated rx -179.15 ry 0 rz -30.08 deg; joints [-2.642, -66.385, 121.4, -183.637, 54.877, 242.218]
  MoveL 5095 to (-315.54, 7.25, -288.53) mm, rotated rx -179.15 ry 0 rz -30.08 deg; joints [-2.642, -66.385, 121.4, -183.637, 54.877, 242.218]
  MoveL 5096 to (-315.54, 7.25, -291.07) mm, rotated rx -179.15 ry 0 rz -30.08 deg; joints [-2.637, -66.253, 121.195, -183.635, 54.805, 242.22]
  MoveC 5097 to (-315.82, 6.77, -292.42) mm, rotated rx -179.15 ry 0 rz -30.08 deg; joints [-2.646, -66.158, 121.094, -183.647, 54.799, 242.227] to (-316.49, 5.6, -292.97) mm, rotated rx -179.15 ry 0 rz -30.08 deg; joints [-2.675, -66.069, 121.068, -183.679, 54.863, 242.242]
  MoveL 5098 to (-316.49, 5.6, -292.97) mm, rotated rx -179.15 ry 0 rz -30.08 deg; joints [-2.675, -66.069, 121.068, -183.679, 54.863, 242.242]
  MoveC 5099 to (-316.55, 5.47, -292.97) mm, rotated rx -179.15 ry 0 rz -30.08 deg; joints [-2.678, -66.062, 121.07, -183.682, 54.872, 242.243] to (-316.58, 5.33, -292.97) mm, rotated rx -179.15 ry 0 rz -30.08 deg; joints [-2.679, -66.055, 121.072, -183.683, 54.881, 242.243]
  MoveL 5100 to (-316.58, 5.33, -292.97) mm, rotated rx -179.15 ry 0 rz -30.08 deg; joints [-2.679, -66.055, 121.072, -183.683, 54.881, 242.243]
  MoveC 5101 to (-316.6, 5.18, -292.97) mm, rotated rx -179.15 ry 0 rz -30.08 deg; joints [-2.68, -66.048, 121.074, -183.684, 54.891, 242.243] to (-316.66, 5.05, -292.97) mm, rotated rx -179.15 ry 0 rz -30.08 deg; joints [-2.683, -66.041, 121.077, -183.687, 54.9, 242.245]
  MoveL 5102 to (-316.66, 5.05, -292.97) mm, rotated rx -179.15 ry 0 rz -30.08 deg; joints [-2.683, -66.041, 121.077, -183.687, 54.9, 242.245]
  MoveL 5103 to (-327.16, -13.08, -292.97) mm, rotated rx -179.15 ry 0 rz -30.08 deg; joints [-3.148, -65.092, 121.341, -184.194, 56.129, 242.461]
  MoveC 5104 to (-327.25, -13.19, -292.97) mm, rotated rx -179.15 ry 0 rz -30.08 deg; joints [-3.152, -65.085, 121.342, -184.198, 56.137, 242.463] to (-327.36, -13.29, -292.97) mm, rotated rx -179.15 ry 0 rz -30.08 deg; joints [-3.157, -65.08, 121.343, -184.204, 56.143, 242.466]
  MoveL 5105 to (-327.36, -13.29, -292.97) mm, rotated rx -179.15 ry 0 rz -30.08 deg; joints [-3.157, -65.08, 121.343, -184.204, 56.143, 242.466]
  MoveC 5106 to (-327.47, -13.38, -292.97) mm, rotated rx -179.15 ry 0 rz -30.08 deg; joints [-3.162, -65.075, 121.344, -184.209, 56.149, 242.469] to (-327.55, -13.5, -292.97) mm, rotated rx -179.15 ry 0 rz -30.08 deg; joints [-3.166, -65.069, 121.346, -184.213, 56.157, 242.471]
  MoveL 5107 to (-327.55, -13.5, -292.97) mm, rotated rx -179.15 ry 0 rz -30.08 deg; joints [-3.166, -65.069, 121.346, -184.213, 56.157, 242.471]
  MoveC 5108 to (-328.23, -14.66, -293.53) mm, rotated rx -179.15 ry 0 rz -30.08 deg; joints [-3.194, -64.979, 121.316, -184.245, 56.219, 242.484] to (-328.51, -15.14, -294.88) mm, rotated rx -179.15 ry 0 rz -30.08 deg; joints [-3.203, -64.885, 121.214, -184.256, 56.211, 242.491]
  MoveL 5109 to (-328.51, -15.14, -294.88) mm, rotated rx -179.15 ry 0 rz -30.08 deg; joints [-3.203, -64.885, 121.214, -184.256, 56.211, 242.491]
  MoveL 5110 to (-328.51, -15.14, -297.42) mm, rotated rx -179.15 ry 0 rz -30.08 deg; joints [-3.197, -64.756, 121.008, -184.253, 56.134, 242.494]
  MoveC 5111 to (-328.23, -14.66, -298.76) mm, rotated rx -179.15 ry 0 rz -30.08 deg; joints [-3.182, -64.713, 120.893, -184.238, 56.061, 242.49] to (-327.55, -13.5, -299.32) mm, rotated rx -179.15 ry 0 rz -30.08 deg; joints [-3.151, -64.746, 120.832, -184.205, 55.966, 242.477]
  MoveL 5112 to (-327.55, -13.5, -299.32) mm, rotated rx -179.15 ry 0 rz -30.08 deg; joints [-3.151, -64.746, 120.832, -184.205, 55.966, 242.477]
  MoveC 5113 to (-327.47, -13.38, -299.32) mm, rotated rx -179.15 ry 0 rz -30.08 deg; joints [-3.147, -64.753, 120.83, -184.201, 55.958, 242.476] to (-327.36, -13.29, -299.32) mm, rotated rx -179.15 ry 0 rz -30.08 deg; joints [-3.142, -64.758, 120.829, -184.195, 55.952, 242.473]
  MoveL 5114 to (-327.36, -13.29, -299.32) mm, rotated rx -179.15 ry 0 rz -30.08 deg; joints [-3.142, -64.758, 120.829, -184.195, 55.952, 242.473]
  MoveC 5115 to (-327.25, -13.19, -299.32) mm, rotated rx -179.15 ry 0 rz -30.08 deg; joints [-3.137, -64.763, 120.828, -184.189, 55.945, 242.47] to (-327.16, -13.08, -299.32) mm, rotated rx -179.15 ry 0 rz -30.08 deg; joints [-3.133, -64.769, 120.827, -184.185, 55.938, 242.468]
  MoveL 5116 to (-327.16, -13.08, -299.32) mm, rotated rx -179.15 ry 0 rz -30.08 deg; joints [-3.133, -64.769, 120.827, -184.185, 55.938, 242.468]
